Yaskawa INFORM job: A_ROOF_UPPER_0614_2_PAINT_47.JBI

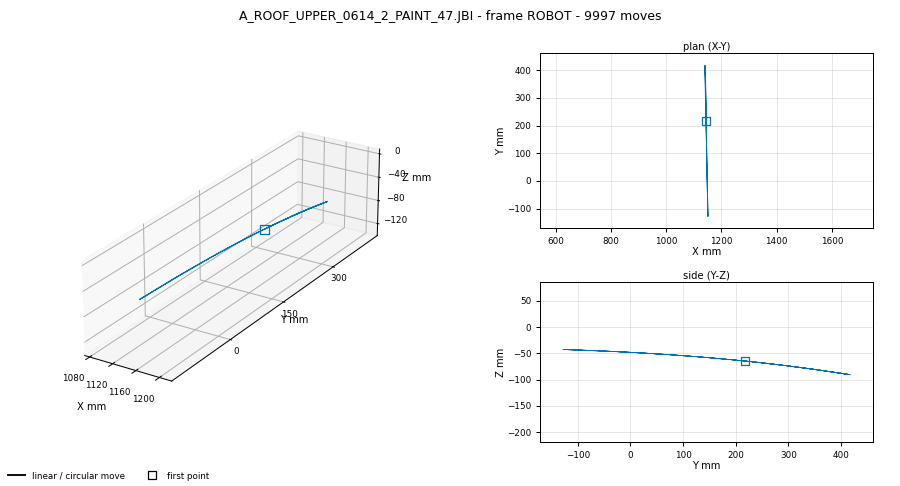
[picture p0: tool path of A_ROOF_UPPER_0614_2_PAINT_47.JBI in frame ROBOT, 9997 of 9997 moves have a stored position in this frame; points joined in program order, loops and branches not executed]
/JOB
//NAME A_ROOF_UPPER_0614_2_PAINT47
//POS
///NPOS 9997,0,0,0,0,0
///TOOL 1
///USER 0
///POSTYPE ROBOT
///RECTAN
///RCONF 1,0,0,0,0,0,0,0,0,0,0,0,0,0,0,0,0,0,0,0,0,0,0,0
C00000=1145.413,218.095,-64.507,-177.907,7.562,148.827
C00001=1145.408,218.343,-64.532,-177.904,7.565,148.827
C00002=1145.404,218.592,-64.557,-177.901,7.567,148.827
C00003=1145.399,218.840,-64.583,-177.899,7.570,148.827
C00004=1145.395,219.089,-64.609,-177.896,7.572,148.827
C00005=1145.391,219.338,-64.634,-177.893,7.575,148.827
C00006=1145.385,219.587,-64.659,-177.890,7.578,148.826
C00007=1145.381,219.835,-64.685,-177.888,7.580,148.826
C00008=1145.377,220.084,-64.711,-177.885,7.583,148.826
C00009=1145.372,220.332,-64.736,-177.882,7.586,148.826
C00010=1145.368,220.581,-64.762,-177.879,7.588,148.826
C00011=1145.364,220.830,-64.787,-177.877,7.591,148.825
C00012=1145.359,221.079,-64.812,-177.874,7.593,148.825
C00013=1145.354,221.327,-64.838,-177.871,7.596,148.825
C00014=1145.350,221.576,-64.864,-177.868,7.599,148.825
C00015=1145.345,221.824,-64.889,-177.865,7.602,148.825
C00016=1145.341,222.073,-64.915,-177.863,7.604,148.825
C00017=1145.337,222.322,-64.940,-177.860,7.607,148.825
C00018=1145.332,222.570,-64.966,-177.857,7.609,148.824
C00019=1145.328,222.819,-64.992,-177.854,7.612,148.824
C00020=1145.324,223.068,-65.017,-177.852,7.614,148.824
C00021=1145.319,223.316,-65.043,-177.849,7.617,148.824
C00022=1145.314,223.565,-65.068,-177.846,7.620,148.824
C00023=1145.310,223.813,-65.094,-177.843,7.623,148.824
C00024=1145.305,224.062,-65.121,-177.840,7.626,148.824
C00025=1145.300,224.311,-65.146,-177.838,7.628,148.823
C00026=1145.296,224.559,-65.172,-177.835,7.631,148.823
C00027=1145.292,224.808,-65.197,-177.832,7.634,148.823
C00028=1145.287,225.056,-65.223,-177.829,7.636,148.823
C00029=1145.283,225.305,-65.249,-177.826,7.639,148.823
C00030=1145.278,225.554,-65.275,-177.824,7.641,148.823
C00031=1145.274,225.803,-65.301,-177.821,7.644,148.823
C00032=1145.270,226.051,-65.327,-177.818,7.647,148.823
C00033=1145.265,226.299,-65.353,-177.815,7.650,148.822
C00034=1145.261,226.548,-65.378,-177.812,7.653,148.822
C00035=1145.256,226.797,-65.405,-177.809,7.656,148.822
C00036=1145.252,227.046,-65.430,-177.807,7.658,148.822
C00037=1145.247,227.294,-65.456,-177.804,7.661,148.822
C00038=1145.243,227.542,-65.482,-177.801,7.663,148.822
C00039=1145.239,227.791,-65.508,-177.798,7.666,148.822
C00040=1145.234,228.040,-65.534,-177.796,7.669,148.821
C00041=1145.229,228.289,-65.560,-177.793,7.671,148.821
C00042=1145.226,228.537,-65.587,-177.791,7.674,148.821
C00043=1145.220,228.786,-65.613,-177.788,7.677,148.821
C00044=1145.216,229.034,-65.638,-177.785,7.679,148.821
C00045=1145.212,229.283,-65.665,-177.782,7.682,148.821
C00046=1145.208,229.531,-65.691,-177.779,7.685,148.821
C00047=1145.203,229.781,-65.717,-177.776,7.688,148.821
C00048=1145.199,230.029,-65.743,-177.774,7.690,148.820
C00049=1145.194,230.277,-65.769,-177.771,7.693,148.820
C00050=1145.189,230.526,-65.795,-177.768,7.696,148.820
C00051=1145.185,230.774,-65.822,-177.765,7.699,148.820
C00052=1145.181,231.023,-65.847,-177.762,7.702,148.820
C00053=1145.176,231.272,-65.874,-177.760,7.705,148.820
C00054=1145.172,231.520,-65.900,-177.757,7.707,148.820
C00055=1145.167,231.769,-65.926,-177.755,7.710,148.820
C00056=1145.163,232.018,-65.953,-177.752,7.713,148.820
C00057=1145.158,232.266,-65.978,-177.748,7.715,148.819
C00058=1145.154,232.514,-66.005,-177.746,7.718,148.819
C00059=1145.149,232.763,-66.031,-177.743,7.721,148.819
C00060=1145.145,233.011,-66.058,-177.740,7.724,148.819
C00061=1145.140,233.260,-66.084,-177.738,7.726,148.819
C00062=1145.136,233.509,-66.111,-177.735,7.729,148.819
C00063=1145.132,233.758,-66.137,-177.732,7.732,148.819
C00064=1145.128,234.006,-66.163,-177.730,7.735,148.819
C00065=1145.123,234.255,-66.190,-177.726,7.737,148.818
C00066=1145.119,234.503,-66.216,-177.723,7.740,148.818
C00067=1145.114,234.751,-66.243,-177.721,7.743,148.818
C00068=1145.110,235.000,-66.269,-177.718,7.746,148.818
C00069=1145.105,235.272,-66.298,-177.715,7.749,148.818
C00070=1145.099,235.544,-66.327,-177.712,7.752,148.818
C00071=1145.095,235.815,-66.356,-177.709,7.754,148.818
C00072=1145.090,236.088,-66.385,-177.706,7.758,148.818
C00073=1145.086,236.336,-66.412,-177.703,7.760,148.817
C00074=1145.082,236.585,-66.438,-177.701,7.763,148.817
C00075=1145.077,236.834,-66.465,-177.698,7.766,148.817
C00076=1145.073,237.082,-66.492,-177.695,7.769,148.817
C00077=1145.068,237.331,-66.518,-177.692,7.772,148.817
C00078=1145.064,237.579,-66.544,-177.689,7.775,148.817
C00079=1145.059,237.827,-66.571,-177.687,7.778,148.817
C00080=1145.055,238.076,-66.599,-177.684,7.781,148.817
C00081=1145.051,238.325,-66.624,-177.681,7.783,148.817
C00082=1145.046,238.573,-66.651,-177.678,7.785,148.816
C00083=1145.041,238.822,-66.678,-177.676,7.788,148.816
C00084=1145.037,239.070,-66.705,-177.673,7.791,148.816
C00085=1145.033,239.318,-66.732,-177.670,7.794,148.816
C00086=1145.028,239.567,-66.759,-177.667,7.797,148.816
C00087=1145.024,239.816,-66.785,-177.664,7.800,148.816
C00088=1145.019,240.064,-66.812,-177.662,7.803,148.816
C00089=1145.014,240.313,-66.839,-177.659,7.806,148.816
C00090=1145.011,240.561,-66.865,-177.656,7.809,148.816
C00091=1145.006,240.809,-66.892,-177.653,7.812,148.816
C00092=1145.002,241.059,-66.920,-177.651,7.815,148.816
C00093=1144.998,241.307,-66.946,-177.648,7.818,148.816
C00094=1144.993,241.555,-66.973,-177.646,7.820,148.816
C00095=1144.989,241.804,-67.000,-177.643,7.823,148.815
C00096=1144.984,242.052,-67.028,-177.640,7.826,148.815
C00097=1144.980,242.300,-67.054,-177.637,7.828,148.815
C00098=1144.975,242.549,-67.081,-177.634,7.831,148.815
C00099=1144.971,242.797,-67.108,-177.631,7.834,148.815
C00100=1144.967,243.047,-67.136,-177.628,7.837,148.815
C00101=1144.962,243.295,-67.163,-177.626,7.840,148.815
C00102=1144.958,243.543,-67.189,-177.623,7.843,148.815
C00103=1144.953,243.792,-67.216,-177.620,7.846,148.815
C00104=1144.949,244.040,-67.243,-177.617,7.849,148.815
C00105=1144.944,244.289,-67.270,-177.614,7.852,148.814
C00106=1144.940,244.537,-67.298,-177.612,7.854,148.814
C00107=1144.936,244.786,-67.325,-177.609,7.857,148.814
C00108=1144.932,245.034,-67.352,-177.606,7.860,148.814
C00109=1144.927,245.283,-67.379,-177.603,7.863,148.814
C00110=1144.922,245.531,-67.406,-177.601,7.865,148.814
C00111=1144.918,245.780,-67.433,-177.598,7.868,148.814
C00112=1144.914,246.028,-67.461,-177.595,7.871,148.814
C00113=1144.909,246.277,-67.488,-177.593,7.874,148.814
C00114=1144.905,246.525,-67.515,-177.590,7.877,148.814
C00115=1144.900,246.774,-67.542,-177.587,7.880,148.814
C00116=1144.896,247.022,-67.569,-177.584,7.883,148.814
C00117=1144.892,247.270,-67.597,-177.581,7.886,148.814
C00118=1144.888,247.519,-67.624,-177.579,7.889,148.813
C00119=1144.883,247.767,-67.651,-177.576,7.892,148.813
C00120=1144.879,248.015,-67.679,-177.573,7.895,148.813
C00121=1144.875,248.264,-67.706,-177.570,7.897,148.813
C00122=1144.870,248.513,-67.733,-177.568,7.900,148.813
C00123=1144.866,248.761,-67.761,-177.565,7.903,148.813
C00124=1144.861,249.009,-67.788,-177.562,7.906,148.813
C00125=1144.857,249.259,-67.816,-177.559,7.909,148.813
C00126=1144.853,249.506,-67.843,-177.556,7.912,148.813
C00127=1144.848,249.755,-67.871,-177.554,7.915,148.813
C00128=1144.844,250.003,-67.899,-177.551,7.918,148.813
C00129=1144.840,250.252,-67.926,-177.548,7.921,148.813
C00130=1144.835,250.500,-67.953,-177.546,7.924,148.813
C00131=1144.831,250.748,-67.981,-177.543,7.927,148.813
C00132=1144.827,250.998,-68.008,-177.540,7.930,148.813
C00133=1144.822,251.245,-68.036,-177.537,7.933,148.813
C00134=1144.817,251.494,-68.063,-177.535,7.936,148.813
C00135=1144.813,251.743,-68.092,-177.532,7.939,148.812
C00136=1144.808,251.991,-68.119,-177.529,7.942,148.812
C00137=1144.804,252.239,-68.146,-177.526,7.945,148.812
C00138=1144.800,252.488,-68.175,-177.523,7.948,148.812
C00139=1144.796,252.736,-68.202,-177.521,7.950,148.812
C00140=1144.791,252.984,-68.229,-177.518,7.953,148.812
C00141=1144.787,253.233,-68.257,-177.515,7.956,148.812
C00142=1144.783,253.481,-68.285,-177.512,7.959,148.812
C00143=1144.778,253.730,-68.313,-177.509,7.962,148.812
C00144=1144.774,253.979,-68.340,-177.507,7.965,148.812
C00145=1144.769,254.226,-68.368,-177.504,7.968,148.812
C00146=1144.766,254.475,-68.396,-177.501,7.971,148.812
C00147=1144.761,254.724,-68.423,-177.499,7.974,148.812
C00148=1144.756,254.972,-68.452,-177.496,7.977,148.812
C00149=1144.752,255.220,-68.480,-177.493,7.980,148.812
C00150=1144.747,255.469,-68.507,-177.490,7.983,148.812
C00151=1144.744,255.717,-68.535,-177.488,7.986,148.812
C00152=1144.739,255.966,-68.563,-177.485,7.989,148.812
C00153=1144.735,256.214,-68.592,-177.482,7.992,148.811
C00154=1144.730,256.463,-68.619,-177.479,7.995,148.811
C00155=1144.726,256.710,-68.646,-177.476,7.998,148.811
C00156=1144.721,256.959,-68.675,-177.474,8.001,148.811
C00157=1144.717,257.207,-68.703,-177.471,8.004,148.811
C00158=1144.713,257.456,-68.731,-177.469,8.007,148.811
C00159=1144.709,257.704,-68.758,-177.466,8.010,148.811
C00160=1144.704,257.953,-68.787,-177.463,8.013,148.811
C00161=1144.700,258.201,-68.815,-177.460,8.015,148.811
C00162=1144.696,258.450,-68.843,-177.457,8.018,148.811
C00163=1144.691,258.698,-68.871,-177.455,8.021,148.811
C00164=1144.687,258.946,-68.899,-177.452,8.024,148.811
C00165=1144.683,259.194,-68.927,-177.449,8.028,148.811
C00166=1144.678,259.443,-68.956,-177.447,8.030,148.811
C00167=1144.674,259.691,-68.984,-177.444,8.033,148.811
C00168=1144.669,259.940,-69.012,-177.441,8.036,148.811
C00169=1144.665,260.188,-69.040,-177.438,8.039,148.811
C00170=1144.661,260.436,-69.068,-177.436,8.042,148.811
C00171=1144.656,260.685,-69.097,-177.432,8.046,148.811
C00172=1144.653,260.933,-69.125,-177.430,8.049,148.811
C00173=1144.647,261.207,-69.156,-177.427,8.052,148.811
C00174=1144.642,261.480,-69.187,-177.424,8.056,148.811
C00175=1144.638,261.753,-69.217,-177.421,8.059,148.811
C00176=1144.633,262.028,-69.249,-177.418,8.062,148.811
C00177=1144.629,262.275,-69.278,-177.415,8.065,148.811
C00178=1144.624,262.524,-69.306,-177.412,8.068,148.811
C00179=1144.620,262.772,-69.334,-177.409,8.071,148.811
C00180=1144.616,263.021,-69.363,-177.406,8.074,148.810
C00181=1144.611,263.269,-69.391,-177.404,8.077,148.811
C00182=1144.607,263.518,-69.419,-177.401,8.080,148.811
C00183=1144.603,263.766,-69.447,-177.398,8.083,148.811
C00184=1144.598,264.014,-69.477,-177.396,8.086,148.810
C00185=1144.595,264.262,-69.505,-177.393,8.089,148.810
C00186=1144.589,264.510,-69.533,-177.391,8.092,148.811
C00187=1144.586,264.759,-69.561,-177.388,8.095,148.810
C00188=1144.581,265.008,-69.590,-177.385,8.098,148.810
C00189=1144.576,265.255,-69.619,-177.382,8.101,148.810
C00190=1144.573,265.504,-69.647,-177.379,8.104,148.810
C00191=1144.568,265.752,-69.676,-177.377,8.108,148.810
C00192=1144.564,266.000,-69.704,-177.374,8.111,148.810
C00193=1144.560,266.249,-69.733,-177.371,8.114,148.810
C00194=1144.555,266.497,-69.762,-177.368,8.117,148.810
C00195=1144.551,266.745,-69.790,-177.365,8.120,148.810
C00196=1144.547,266.994,-69.819,-177.363,8.123,148.810
C00197=1144.542,267.242,-69.847,-177.360,8.126,148.810
C00198=1144.538,267.490,-69.876,-177.357,8.129,148.810
C00199=1144.534,267.739,-69.905,-177.355,8.132,148.810
C00200=1144.529,267.987,-69.933,-177.352,8.135,148.810
C00201=1144.525,268.235,-69.962,-177.350,8.138,148.810
C00202=1144.521,268.484,-69.991,-177.346,8.142,148.810
C00203=1144.516,268.732,-70.020,-177.343,8.145,148.810
C00204=1144.512,268.980,-70.048,-177.341,8.148,148.810
C00205=1144.508,269.229,-70.078,-177.338,8.151,148.810
C00206=1144.503,269.477,-70.106,-177.336,8.154,148.810
C00207=1144.499,269.725,-70.135,-177.333,8.157,148.810
C00208=1144.495,269.974,-70.164,-177.330,8.160,148.810
C00209=1144.491,270.222,-70.193,-177.328,8.163,148.810
C00210=1144.486,270.471,-70.222,-177.325,8.166,148.810
C00211=1144.482,270.718,-70.250,-177.321,8.170,148.810
C00212=1144.478,270.967,-70.279,-177.319,8.173,148.810
C00213=1144.473,271.215,-70.309,-177.316,8.176,148.810
C00214=1144.469,271.463,-70.338,-177.314,8.179,148.810
C00215=1144.464,271.712,-70.366,-177.311,8.182,148.810
C00216=1144.461,271.960,-70.395,-177.308,8.185,148.810
C00217=1144.457,272.208,-70.425,-177.306,8.188,148.810
C00218=1144.452,272.457,-70.453,-177.303,8.191,148.810
C00219=1144.447,272.704,-70.483,-177.300,8.194,148.810
C00220=1144.443,272.953,-70.512,-177.297,8.198,148.810
C00221=1144.439,273.201,-70.541,-177.294,8.201,148.810
C00222=1144.434,273.450,-70.570,-177.292,8.204,148.810
C00223=1144.431,273.698,-70.599,-177.289,8.207,148.810
C00224=1144.426,273.946,-70.627,-177.287,8.210,148.810
C00225=1144.422,274.194,-70.657,-177.284,8.213,148.810
C00226=1144.418,274.442,-70.686,-177.281,8.216,148.811
C00227=1144.413,274.691,-70.716,-177.278,8.220,148.811
C00228=1144.409,274.939,-70.745,-177.275,8.223,148.810
C00229=1144.405,275.188,-70.774,-177.273,8.226,148.811
C00230=1144.401,275.436,-70.803,-177.270,8.229,148.811
C00231=1144.396,275.684,-70.833,-177.267,8.232,148.811
C00232=1144.392,275.932,-70.862,-177.265,8.235,148.810
C00233=1144.387,276.180,-70.891,-177.262,8.238,148.811
C00234=1144.383,276.428,-70.921,-177.259,8.242,148.811
C00235=1144.379,276.677,-70.950,-177.256,8.245,148.811
C00236=1144.376,276.925,-70.979,-177.254,8.248,148.811
C00237=1144.371,277.174,-71.008,-177.251,8.251,148.811
C00238=1144.367,277.422,-71.037,-177.248,8.254,148.811
C00239=1144.362,277.669,-71.066,-177.246,8.257,148.811
C00240=1144.357,277.918,-71.097,-177.243,8.261,148.811
C00241=1144.353,278.166,-71.126,-177.240,8.264,148.811
C00242=1144.349,278.414,-71.155,-177.237,8.267,148.811
C00243=1144.345,278.663,-71.185,-177.235,8.270,148.811
C00244=1144.340,278.911,-71.214,-177.232,8.273,148.811
C00245=1144.336,279.159,-71.244,-177.229,8.276,148.811
C00246=1144.332,279.408,-71.273,-177.226,8.280,148.811
C00247=1144.328,279.656,-71.303,-177.224,8.283,148.811
C00248=1144.324,279.903,-71.333,-177.221,8.286,148.811
C00249=1144.320,280.152,-71.362,-177.218,8.289,148.811
C00250=1144.316,280.400,-71.392,-177.216,8.293,148.811
C00251=1144.312,280.648,-71.421,-177.213,8.295,148.811
C00252=1144.307,280.897,-71.451,-177.210,8.300,148.811
C00253=1144.302,281.145,-71.481,-177.207,8.302,148.811
C00254=1144.298,281.393,-71.510,-177.205,8.305,148.811
C00255=1144.294,281.642,-71.540,-177.202,8.309,148.811
C00256=1144.290,281.889,-71.570,-177.200,8.312,148.811
C00257=1144.286,282.138,-71.599,-177.197,8.316,148.812
C00258=1144.281,282.386,-71.629,-177.194,8.319,148.811
C00259=1144.277,282.634,-71.659,-177.191,8.322,148.811
C00260=1144.273,282.882,-71.689,-177.189,8.325,148.812
C00261=1144.269,283.130,-71.718,-177.186,8.328,148.812
C00262=1144.265,283.379,-71.748,-177.184,8.331,148.812
C00263=1144.260,283.627,-71.778,-177.180,8.335,148.812
C00264=1144.256,283.875,-71.808,-177.178,8.338,148.812
C00265=1144.252,284.123,-71.837,-177.175,8.341,148.812
C00266=1144.248,284.371,-71.867,-177.172,8.344,148.812
C00267=1144.243,284.619,-71.898,-177.170,8.347,148.812
C00268=1144.239,284.868,-71.927,-177.167,8.351,148.812
C00269=1144.235,285.116,-71.957,-177.164,8.354,148.812
C00270=1144.230,285.364,-71.987,-177.162,8.357,148.812
C00271=1144.226,285.612,-72.017,-177.159,8.360,148.812
C00272=1144.222,285.860,-72.047,-177.156,8.364,148.812
C00273=1144.217,286.108,-72.077,-177.154,8.367,148.812
C00274=1144.213,286.357,-72.106,-177.151,8.370,148.812
C00275=1144.209,286.604,-72.137,-177.148,8.373,148.812
C00276=1144.205,286.854,-72.167,-177.146,8.376,148.812
C00277=1144.200,287.128,-72.200,-177.142,8.380,148.812
C00278=1144.195,287.403,-72.234,-177.139,8.384,148.813
C00279=1144.191,287.679,-72.267,-177.137,8.387,148.813
C00280=1144.186,287.954,-72.301,-177.134,8.391,148.813
C00281=1144.182,288.203,-72.330,-177.131,8.394,148.813
C00282=1144.177,288.451,-72.361,-177.128,8.398,148.813
C00283=1144.173,288.699,-72.391,-177.125,8.401,148.813
C00284=1144.169,288.947,-72.421,-177.123,8.405,148.813
C00285=1144.165,289.195,-72.452,-177.120,8.407,148.813
C00286=1144.161,289.443,-72.481,-177.117,8.412,148.813
C00287=1144.156,289.691,-72.512,-177.114,8.415,148.813
C00288=1144.153,289.940,-72.542,-177.112,8.418,148.813
C00289=1144.148,290.188,-72.572,-177.109,8.421,148.813
C00290=1144.144,290.436,-72.603,-177.107,8.424,148.814
C00291=1144.139,290.684,-72.633,-177.104,8.428,148.814
C00292=1144.135,290.932,-72.663,-177.101,8.431,148.814
C00293=1144.131,291.181,-72.694,-177.098,8.434,148.814
C00294=1144.127,291.428,-72.724,-177.096,8.437,148.814
C00295=1144.123,291.676,-72.755,-177.093,8.441,148.814
C00296=1144.118,291.925,-72.784,-177.090,8.444,148.814
C00297=1144.114,292.173,-72.815,-177.088,8.447,148.814
C00298=1144.110,292.421,-72.846,-177.085,8.450,148.814
C00299=1144.106,292.669,-72.876,-177.082,8.454,148.814
C00300=1144.102,292.916,-72.907,-177.080,8.457,148.814
C00301=1144.097,293.165,-72.937,-177.077,8.461,148.814
C00302=1144.094,293.413,-72.967,-177.075,8.464,148.814
C00303=1144.089,293.661,-72.998,-177.072,8.468,148.815
C00304=1144.085,293.909,-73.029,-177.069,8.471,148.815
C00305=1144.081,294.157,-73.059,-177.066,8.474,148.815
C00306=1144.077,294.406,-73.090,-177.063,8.478,148.815
C00307=1144.072,294.654,-73.121,-177.061,8.481,148.815
C00308=1144.068,294.901,-73.151,-177.058,8.484,148.815
C00309=1144.064,295.150,-73.182,-177.056,8.487,148.815
C00310=1144.060,295.398,-73.212,-177.053,8.491,148.815
C00311=1144.056,295.645,-73.243,-177.050,8.494,148.815
C00312=1144.051,295.894,-73.273,-177.048,8.497,148.815
C00313=1144.047,296.142,-73.303,-177.045,8.501,148.816
C00314=1144.043,296.390,-73.335,-177.042,8.504,148.816
C00315=1144.039,296.638,-73.366,-177.040,8.508,148.816
C00316=1144.035,296.886,-73.397,-177.037,8.511,148.816
C00317=1144.031,297.134,-73.427,-177.034,8.515,148.816
C00318=1144.026,297.382,-73.458,-177.032,8.518,148.816
C00319=1144.022,297.631,-73.489,-177.029,8.521,148.816
C00320=1144.018,297.878,-73.519,-177.026,8.524,148.816
C00321=1144.014,298.126,-73.550,-177.023,8.528,148.816
C00322=1144.010,298.375,-73.581,-177.021,8.531,148.816
C00323=1144.005,298.623,-73.612,-177.018,8.534,148.817
C00324=1144.001,298.872,-73.643,-177.015,8.538,148.817
C00325=1143.997,299.119,-73.674,-177.013,8.541,148.817
C00326=1143.993,299.366,-73.705,-177.010,8.545,148.817
C00327=1143.989,299.615,-73.736,-177.007,8.548,148.817
C00328=1143.984,299.863,-73.766,-177.005,8.552,148.817
C00329=1143.980,300.111,-73.797,-177.002,8.555,148.817
C00330=1143.976,300.359,-73.829,-177.000,8.558,148.817
C00331=1143.972,300.607,-73.859,-176.997,8.562,148.818
C00332=1143.968,300.855,-73.890,-176.994,8.565,148.818
C00333=1143.964,301.103,-73.922,-176.992,8.568,148.818
C00334=1143.960,301.351,-73.953,-176.989,8.572,148.818
C00335=1143.955,301.599,-73.984,-176.986,8.576,148.818
C00336=1143.950,301.847,-74.014,-176.984,8.578,148.818
C00337=1143.947,302.095,-74.046,-176.981,8.583,148.818
C00338=1143.942,302.343,-74.077,-176.978,8.586,148.818
C00339=1143.938,302.591,-74.109,-176.976,8.589,148.818
C00340=1143.934,302.839,-74.140,-176.973,8.593,148.819
C00341=1143.930,303.088,-74.170,-176.970,8.596,148.819
C00342=1143.926,303.335,-74.202,-176.968,8.599,148.819
C00343=1143.922,303.583,-74.232,-176.965,8.603,148.819
C00344=1143.918,303.831,-74.264,-176.962,8.606,148.819
C00345=1143.913,304.079,-74.295,-176.960,8.610,148.819
C00346=1143.909,304.328,-74.326,-176.957,8.613,148.819
C00347=1143.905,304.575,-74.358,-176.954,8.617,148.819
C00348=1143.901,304.824,-74.389,-176.952,8.620,148.820
C00349=1143.897,305.071,-74.420,-176.949,8.624,148.820
C00350=1143.893,305.320,-74.451,-176.946,8.627,148.820
C00351=1143.888,305.567,-74.483,-176.944,8.630,148.820
C00352=1143.884,305.815,-74.515,-176.941,8.634,148.820
C00353=1143.879,306.063,-74.546,-176.939,8.638,148.820
C00354=1143.875,306.311,-74.578,-176.936,8.640,148.820
C00355=1143.871,306.559,-74.609,-176.933,8.645,148.821
C00356=1143.867,306.807,-74.641,-176.931,8.648,148.821
C00357=1143.863,307.055,-74.672,-176.928,8.651,148.821
C00358=1143.859,307.303,-74.703,-176.925,8.655,148.821
C00359=1143.855,307.551,-74.735,-176.923,8.658,148.821
C00360=1143.851,307.799,-74.766,-176.920,8.661,148.821
C00361=1143.847,308.047,-74.798,-176.917,8.665,148.822
C00362=1143.843,308.295,-74.829,-176.915,8.669,148.822
C00363=1143.838,308.543,-74.862,-176.912,8.672,148.822
C00364=1143.834,308.792,-74.893,-176.909,8.676,148.822
C00365=1143.830,309.039,-74.924,-176.907,8.679,148.822
C00366=1143.826,309.287,-74.956,-176.904,8.683,148.822
C00367=1143.822,309.534,-74.987,-176.901,8.686,148.822
C00368=1143.818,309.783,-75.019,-176.899,8.689,148.822
C00369=1143.813,310.031,-75.051,-176.896,8.693,148.823
C00370=1143.809,310.279,-75.083,-176.894,8.697,148.823
C00371=1143.805,310.527,-75.114,-176.891,8.700,148.823
C00372=1143.801,310.774,-75.146,-176.888,8.704,148.823
C00373=1143.797,311.022,-75.178,-176.886,8.707,148.823
C00374=1143.793,311.271,-75.209,-176.883,8.711,148.823
C00375=1143.788,311.518,-75.241,-176.880,8.714,148.824
C00376=1143.784,311.767,-75.273,-176.878,8.718,148.824
C00377=1143.780,312.015,-75.305,-176.875,8.722,148.824
C00378=1143.776,312.262,-75.337,-176.873,8.725,148.824
C00379=1143.772,312.510,-75.369,-176.869,8.729,148.824
C00380=1143.768,312.758,-75.400,-176.867,8.732,148.824
C00381=1143.763,313.036,-75.437,-176.864,8.736,148.825
C00382=1143.759,313.314,-75.472,-176.861,8.740,148.825
C00383=1143.754,313.591,-75.508,-176.858,8.744,148.825
C00384=1143.749,313.870,-75.543,-176.855,8.748,148.825
C00385=1143.746,314.117,-75.576,-176.853,8.751,148.826
C00386=1143.741,314.365,-75.608,-176.850,8.754,148.826
C00387=1143.737,314.613,-75.640,-176.847,8.758,148.826
C00388=1143.733,314.861,-75.672,-176.845,8.762,148.826
C00389=1143.729,315.109,-75.704,-176.842,8.766,148.826
C00390=1143.725,315.356,-75.736,-176.840,8.769,148.826
C00391=1143.720,315.605,-75.768,-176.838,8.772,148.827
C00392=1143.717,315.853,-75.800,-176.835,8.776,148.827
C00393=1143.712,316.100,-75.831,-176.832,8.780,148.827
C00394=1143.708,316.348,-75.864,-176.829,8.784,148.827
C00395=1143.704,316.596,-75.896,-176.827,8.787,148.827
C00396=1143.700,316.844,-75.929,-176.824,8.790,148.827
C00397=1143.696,317.092,-75.961,-176.821,8.794,148.828
C00398=1143.691,317.340,-75.993,-176.819,8.797,148.828
C00399=1143.688,317.587,-76.025,-176.816,8.801,148.828
C00400=1143.684,317.835,-76.057,-176.814,8.805,148.828
C00401=1143.680,318.084,-76.089,-176.811,8.809,148.828
C00402=1143.676,318.332,-76.121,-176.809,8.812,148.829
C00403=1143.671,318.579,-76.154,-176.806,8.815,148.829
C00404=1143.667,318.827,-76.186,-176.803,8.819,148.829
C00405=1143.663,319.075,-76.218,-176.801,8.823,148.829
C00406=1143.660,319.323,-76.251,-176.798,8.827,148.829
C00407=1143.655,319.571,-76.283,-176.796,8.830,148.830
C00408=1143.651,319.819,-76.316,-176.793,8.834,148.830
C00409=1143.647,320.066,-76.348,-176.790,8.837,148.830
C00410=1143.642,320.314,-76.380,-176.787,8.841,148.830
C00411=1143.639,320.562,-76.413,-176.785,8.845,148.830
C00412=1143.634,320.810,-76.445,-176.783,8.848,148.831
C00413=1143.631,321.058,-76.478,-176.780,8.852,148.831
C00414=1143.627,321.306,-76.510,-176.778,8.855,148.831
C00415=1143.622,321.554,-76.544,-176.775,8.859,148.831
C00416=1143.618,321.801,-76.575,-176.772,8.863,148.831
C00417=1143.614,322.049,-76.608,-176.769,8.867,148.832
C00418=1143.610,322.297,-76.640,-176.767,8.870,148.832
C00419=1143.606,322.545,-76.673,-176.764,8.874,148.832
C00420=1143.602,322.793,-76.706,-176.762,8.877,148.832
C00421=1143.598,323.040,-76.738,-176.759,8.881,148.832
C00422=1143.594,323.289,-76.771,-176.757,8.885,148.833
C00423=1143.590,323.536,-76.804,-176.754,8.888,148.833
C00424=1143.586,323.784,-76.836,-176.751,8.892,148.833
C00425=1143.582,324.032,-76.869,-176.749,8.895,148.833
C00426=1143.578,324.280,-76.902,-176.746,8.899,148.834
C00427=1143.574,324.528,-76.934,-176.744,8.903,148.834
C00428=1143.570,324.776,-76.967,-176.741,8.907,148.834
C00429=1143.566,325.023,-77.000,-176.738,8.910,148.834
C00430=1143.561,325.271,-77.032,-176.736,8.914,148.834
C00431=1143.557,325.518,-77.065,-176.733,8.917,148.835
C00432=1143.553,325.766,-77.098,-176.730,8.921,148.835
C00433=1143.549,326.014,-77.131,-176.728,8.925,148.835
C00434=1143.545,326.262,-77.164,-176.725,8.929,148.835
C00435=1143.540,326.510,-77.197,-176.723,8.932,148.835
C00436=1143.537,326.757,-77.229,-176.720,8.936,148.836
C00437=1143.533,327.005,-77.262,-176.718,8.940,148.836
C00438=1143.528,327.253,-77.295,-176.715,8.944,148.836
C00439=1143.524,327.501,-77.328,-176.713,8.947,148.836
C00440=1143.520,327.749,-77.361,-176.710,8.951,148.837
C00441=1143.516,327.997,-77.394,-176.707,8.954,148.837
C00442=1143.513,328.244,-77.427,-176.704,8.958,148.837
C00443=1143.509,328.492,-77.460,-176.702,8.962,148.837
C00444=1143.504,328.740,-77.493,-176.699,8.966,148.838
C00445=1143.500,328.987,-77.526,-176.697,8.969,148.838
C00446=1143.496,329.236,-77.559,-176.694,8.973,148.838
C00447=1143.492,329.484,-77.592,-176.692,8.977,148.838
C00448=1143.488,329.732,-77.625,-176.689,8.981,148.839
C00449=1143.484,329.980,-77.659,-176.687,8.984,148.839
C00450=1143.480,330.227,-77.692,-176.684,8.988,148.839
C00451=1143.476,330.475,-77.725,-176.682,8.991,148.839
C00452=1143.472,330.723,-77.758,-176.679,8.995,148.839
C00453=1143.468,330.970,-77.791,-176.677,8.999,148.840
C00454=1143.464,331.218,-77.824,-176.674,9.003,148.840
C00455=1143.460,331.466,-77.857,-176.671,9.006,148.840
C00456=1143.456,331.713,-77.891,-176.669,9.010,148.841
C00457=1143.452,331.960,-77.924,-176.666,9.014,148.841
C00458=1143.448,332.208,-77.957,-176.663,9.018,148.841
C00459=1143.444,332.457,-77.991,-176.661,9.021,148.841
C00460=1143.440,332.704,-78.024,-176.658,9.025,148.842
C00461=1143.436,332.952,-78.057,-176.656,9.029,148.842
C00462=1143.431,333.200,-78.091,-176.653,9.033,148.842
C00463=1143.427,333.448,-78.124,-176.651,9.036,148.842
C00464=1143.423,333.695,-78.158,-176.648,9.040,148.842
C00465=1143.419,333.943,-78.191,-176.646,9.044,148.843
C00466=1143.415,334.191,-78.224,-176.643,9.048,148.843
C00467=1143.411,334.439,-78.258,-176.641,9.051,148.843
C00468=1143.408,334.686,-78.291,-176.638,9.055,148.844
C00469=1143.403,334.934,-78.325,-176.635,9.059,148.844
C00470=1143.399,335.181,-78.358,-176.633,9.063,148.844
C00471=1143.395,335.429,-78.391,-176.630,9.067,148.844
C00472=1143.392,335.677,-78.425,-176.628,9.070,148.845
C00473=1143.387,335.925,-78.459,-176.625,9.074,148.845
C00474=1143.383,336.173,-78.492,-176.623,9.078,148.845
C00475=1143.379,336.420,-78.526,-176.620,9.082,148.846
C00476=1143.375,336.668,-78.559,-176.618,9.085,148.846
C00477=1143.372,336.915,-78.593,-176.615,9.089,148.846
C00478=1143.368,337.163,-78.627,-176.613,9.093,148.846
C00479=1143.363,337.411,-78.660,-176.610,9.097,148.847
C00480=1143.359,337.658,-78.694,-176.607,9.101,148.847
C00481=1143.355,337.907,-78.728,-176.605,9.104,148.847
C00482=1143.351,338.154,-78.762,-176.602,9.109,148.848
C00483=1143.347,338.401,-78.795,-176.600,9.112,148.848
C00484=1143.343,338.649,-78.829,-176.597,9.116,148.848
C00485=1143.339,338.929,-78.867,-176.594,9.120,148.848
C00486=1143.334,339.210,-78.906,-176.592,9.124,148.849
C00487=1143.329,339.491,-78.943,-176.589,9.128,148.849
C00488=1143.325,339.771,-78.981,-176.585,9.133,148.849
C00489=1143.320,340.019,-79.016,-176.583,9.137,148.850
C00490=1143.317,340.267,-79.050,-176.580,9.141,148.850
C00491=1143.313,340.514,-79.083,-176.578,9.144,148.850
C00492=1143.308,340.762,-79.118,-176.575,9.149,148.850
C00493=1143.305,341.010,-79.151,-176.573,9.152,148.851
C00494=1143.301,341.257,-79.185,-176.570,9.156,148.851
C00495=1143.296,341.505,-79.219,-176.568,9.160,148.851
C00496=1143.293,341.753,-79.253,-176.565,9.164,148.852
C00497=1143.288,342.001,-79.287,-176.562,9.168,148.852
C00498=1143.285,342.248,-79.321,-176.561,9.171,148.852
C00499=1143.280,342.495,-79.354,-176.558,9.175,148.852
C00500=1143.276,342.743,-79.389,-176.555,9.179,148.853
C00501=1143.273,342.991,-79.423,-176.553,9.183,148.853
C00502=1143.269,343.239,-79.458,-176.550,9.187,148.853
C00503=1143.265,343.486,-79.491,-176.548,9.190,148.854
C00504=1143.261,343.734,-79.525,-176.545,9.195,148.854
C00505=1143.257,343.982,-79.560,-176.542,9.199,148.854
C00506=1143.253,344.229,-79.594,-176.540,9.202,148.854
C00507=1143.248,344.476,-79.628,-176.537,9.206,148.855
C00508=1143.245,344.724,-79.662,-176.535,9.210,148.855
C00509=1143.240,344.972,-79.696,-176.532,9.214,148.856
C00510=1143.237,345.220,-79.730,-176.530,9.218,148.856
C00511=1143.232,345.467,-79.765,-176.527,9.221,148.856
C00512=1143.229,345.714,-79.799,-176.525,9.226,148.856
C00513=1143.225,345.963,-79.834,-176.522,9.230,148.857
C00514=1143.221,346.210,-79.867,-176.520,9.234,148.857
C00515=1143.217,346.458,-79.902,-176.517,9.238,148.857
C00516=1143.213,346.705,-79.936,-176.515,9.241,148.858
C00517=1143.208,346.952,-79.971,-176.512,9.245,148.858
C00518=1143.204,347.200,-80.005,-176.509,9.249,148.858
C00519=1143.201,347.447,-80.039,-176.507,9.253,148.859
C00520=1143.197,347.696,-80.074,-176.504,9.257,148.859
C00521=1143.193,347.943,-80.108,-176.501,9.261,148.859
C00522=1143.189,348.191,-80.143,-176.500,9.265,148.860
C00523=1143.184,348.438,-80.177,-176.497,9.269,148.860
C00524=1143.181,348.686,-80.212,-176.495,9.272,148.860
C00525=1143.176,348.934,-80.246,-176.492,9.276,148.860
C00526=1143.173,349.181,-80.280,-176.489,9.281,148.861
C00527=1143.169,349.429,-80.315,-176.487,9.284,148.861
C00528=1143.165,349.676,-80.350,-176.484,9.288,148.861
C00529=1143.161,349.923,-80.384,-176.482,9.292,148.862
C00530=1143.157,350.171,-80.419,-176.479,9.296,148.862
C00531=1143.153,350.419,-80.453,-176.477,9.300,148.863
C00532=1143.149,350.667,-80.488,-176.474,9.304,148.863
C00533=1143.145,350.913,-80.523,-176.472,9.308,148.863
C00534=1143.141,351.162,-80.558,-176.469,9.312,148.863
C00535=1143.137,351.409,-80.592,-176.466,9.316,148.864
C00536=1143.133,351.657,-80.626,-176.464,9.320,148.864
C00537=1143.129,351.904,-80.662,-176.462,9.324,148.865
C00538=1143.125,352.152,-80.696,-176.459,9.328,148.865
C00539=1143.121,352.400,-80.731,-176.457,9.332,148.865
C00540=1143.118,352.646,-80.766,-176.454,9.336,148.865
C00541=1143.114,352.894,-80.801,-176.451,9.340,148.866
C00542=1143.109,353.142,-80.835,-176.449,9.343,148.866
C00543=1143.105,353.389,-80.871,-176.446,9.348,148.867
C00544=1143.102,353.637,-80.905,-176.444,9.352,148.867
C00545=1143.098,353.885,-80.939,-176.442,9.355,148.867
C00546=1143.094,354.132,-80.975,-176.439,9.359,148.867
C00547=1143.089,354.380,-81.009,-176.436,9.364,148.868
C00548=1143.086,354.627,-81.045,-176.434,9.367,148.868
C00549=1143.083,354.875,-81.079,-176.431,9.371,148.869
C00550=1143.078,355.122,-81.114,-176.428,9.376,148.869
C00551=1143.074,355.370,-81.149,-176.427,9.379,148.869
C00552=1143.070,355.617,-81.184,-176.424,9.383,148.870
C00553=1143.066,355.865,-81.219,-176.421,9.388,148.870
C00554=1143.062,356.112,-81.255,-176.419,9.391,148.870
C00555=1143.058,356.360,-81.289,-176.416,9.395,148.871
C00556=1143.054,356.607,-81.325,-176.413,9.399,148.871
C00557=1143.051,356.855,-81.359,-176.411,9.403,148.871
C00558=1143.047,357.102,-81.394,-176.409,9.407,148.872
C00559=1143.043,357.349,-81.430,-176.406,9.411,148.872
C00560=1143.039,357.597,-81.465,-176.404,9.416,148.872
C00561=1143.035,357.844,-81.500,-176.401,9.419,148.873
C00562=1143.031,358.092,-81.535,-176.399,9.423,148.873
C00563=1143.027,358.340,-81.570,-176.396,9.427,148.873
C00564=1143.023,358.587,-81.606,-176.394,9.431,148.874
C00565=1143.019,358.834,-81.641,-176.391,9.435,148.874
C00566=1143.015,359.082,-81.676,-176.388,9.440,148.875
C00567=1143.012,359.330,-81.711,-176.386,9.444,148.875
C00568=1143.008,359.577,-81.747,-176.384,9.447,148.875
C00569=1143.004,359.824,-81.782,-176.381,9.452,148.876
C00570=1143.000,360.072,-81.817,-176.378,9.456,148.876
C00571=1142.996,360.320,-81.852,-176.376,9.460,148.876
C00572=1142.992,360.567,-81.888,-176.373,9.463,148.877
C00573=1142.988,360.814,-81.923,-176.371,9.468,148.877
C00574=1142.984,361.061,-81.959,-176.368,9.472,148.877
C00575=1142.981,361.309,-81.994,-176.365,9.476,148.878
C00576=1142.977,361.557,-82.029,-176.363,9.481,148.878
C00577=1142.973,361.804,-82.064,-176.361,9.484,148.878
C00578=1142.968,362.052,-82.100,-176.358,9.488,148.879
C00579=1142.964,362.299,-82.136,-176.355,9.492,148.879
C00580=1142.961,362.547,-82.171,-176.353,9.497,148.880
C00581=1142.957,362.794,-82.207,-176.350,9.501,148.880
C00582=1142.953,363.041,-82.242,-176.347,9.505,148.880
C00583=1142.949,363.288,-82.278,-176.344,9.509,148.881
C00584=1142.946,363.536,-82.313,-176.342,9.513,148.881
C00585=1142.942,363.783,-82.349,-176.340,9.517,148.881
C00586=1142.937,364.031,-82.385,-176.337,9.521,148.882
C00587=1142.934,364.279,-82.420,-176.334,9.526,148.882
C00588=1142.930,364.526,-82.456,-176.331,9.530,148.882
C00589=1142.926,364.810,-82.497,-176.328,9.535,148.883
C00590=1142.921,365.093,-82.538,-176.326,9.539,148.883
C00591=1142.916,365.377,-82.579,-176.322,9.544,148.884
C00592=1142.912,365.660,-82.620,-176.320,9.549,148.884
C00593=1142.908,365.908,-82.655,-176.317,9.553,148.885
C00594=1142.904,366.155,-82.691,-176.314,9.557,148.885
C00595=1142.900,366.403,-82.727,-176.312,9.561,148.885
C00596=1142.897,366.650,-82.763,-176.309,9.565,148.886
C00597=1142.893,366.897,-82.799,-176.306,9.570,148.886
C00598=1142.889,367.145,-82.834,-176.304,9.574,148.886
C00599=1142.885,367.393,-82.870,-176.301,9.578,148.887
C00600=1142.882,367.639,-82.907,-176.299,9.583,148.887
C00601=1142.878,367.887,-82.942,-176.296,9.587,148.888
C00602=1142.873,368.134,-82.978,-176.293,9.591,148.888
C00603=1142.869,368.382,-83.014,-176.290,9.595,148.888
C00604=1142.866,368.628,-83.050,-176.288,9.600,148.889
C00605=1142.861,368.876,-83.086,-176.285,9.604,148.889
C00606=1142.858,369.124,-83.122,-176.282,9.608,148.890
C00607=1142.854,369.371,-83.158,-176.280,9.612,148.890
C00608=1142.850,369.618,-83.194,-176.278,9.616,148.890
C00609=1142.847,369.865,-83.230,-176.275,9.620,148.891
C00610=1142.842,370.113,-83.266,-176.272,9.624,148.891
C00611=1142.839,370.361,-83.302,-176.270,9.629,148.892
C00612=1142.835,370.608,-83.339,-176.267,9.633,148.892
C00613=1142.831,370.855,-83.374,-176.264,9.637,148.892
C00614=1142.827,371.103,-83.411,-176.262,9.642,148.893
C00615=1142.823,371.350,-83.447,-176.259,9.646,148.893
C00616=1142.819,371.597,-83.484,-176.256,9.650,148.894
C00617=1142.815,371.845,-83.519,-176.254,9.655,148.894
C00618=1142.812,372.092,-83.555,-176.251,9.659,148.895
C00619=1142.808,372.339,-83.592,-176.250,9.663,148.895
C00620=1142.804,372.586,-83.628,-176.247,9.667,148.895
C00621=1142.800,372.833,-83.665,-176.244,9.671,148.896
C00622=1142.796,373.081,-83.701,-176.242,9.675,148.896
C00623=1142.792,373.328,-83.737,-176.239,9.680,148.897
C00624=1142.788,373.575,-83.774,-176.237,9.684,148.897
C00625=1142.785,373.823,-83.809,-176.235,9.688,148.897
C00626=1142.781,374.071,-83.847,-176.232,9.692,148.898
C00627=1142.778,374.318,-83.883,-176.230,9.696,148.898
C00628=1142.773,374.565,-83.919,-176.227,9.701,148.899
C00629=1142.770,374.812,-83.955,-176.225,9.704,148.899
C00630=1142.766,375.060,-83.992,-176.223,9.709,148.900
C00631=1142.762,375.307,-84.028,-176.220,9.713,148.900
C00632=1142.758,375.554,-84.065,-176.218,9.718,148.901
C00633=1142.754,375.801,-84.102,-176.216,9.721,148.901
C00634=1142.750,376.049,-84.138,-176.213,9.726,148.902
C00635=1142.747,376.295,-84.175,-176.211,9.729,148.902
C00636=1142.743,376.544,-84.211,-176.209,9.733,148.902
C00637=1142.739,376.791,-84.248,-176.207,9.738,148.903
C00638=1142.735,377.038,-84.284,-176.205,9.742,148.904
C00639=1142.731,377.285,-84.321,-176.202,9.746,148.904
C00640=1142.727,377.532,-84.358,-176.200,9.750,148.904
C00641=1142.724,377.779,-84.394,-176.199,9.754,148.905
C00642=1142.720,378.027,-84.431,-176.196,9.758,148.906
C00643=1142.716,378.275,-84.468,-176.195,9.762,148.906
C00644=1142.713,378.522,-84.504,-176.192,9.766,148.907
C00645=1142.709,378.769,-84.541,-176.190,9.770,148.907
C00646=1142.704,379.016,-84.578,-176.189,9.774,148.908
C00647=1142.700,379.263,-84.614,-176.187,9.778,148.908
C00648=1142.697,379.510,-84.651,-176.185,9.781,148.909
C00649=1142.693,379.758,-84.688,-176.183,9.786,148.909
C00650=1142.689,380.005,-84.725,-176.181,9.789,148.910
C00651=1142.685,380.253,-84.762,-176.180,9.793,148.910
C00652=1142.681,380.500,-84.799,-176.178,9.797,148.911
C00653=1142.678,380.747,-84.835,-176.177,9.801,148.912
C00654=1142.674,380.995,-84.872,-176.176,9.804,148.912
C00655=1142.670,381.242,-84.909,-176.174,9.808,148.913
C00656=1142.666,381.489,-84.946,-176.173,9.812,148.913
C00657=1142.662,381.736,-84.983,-176.171,9.815,148.914
C00658=1142.659,381.982,-85.020,-176.170,9.818,148.914
C00659=1142.656,382.230,-85.057,-176.169,9.822,148.915
C00660=1142.651,382.478,-85.094,-176.167,9.826,148.916
C00661=1142.647,382.725,-85.130,-176.167,9.830,148.916
C00662=1142.643,382.972,-85.167,-176.166,9.833,148.917
C00663=1142.640,383.220,-85.205,-176.164,9.837,148.918
C00664=1142.636,383.467,-85.241,-176.163,9.840,148.918
C00665=1142.633,383.713,-85.278,-176.163,9.843,148.919
C00666=1142.628,383.960,-85.315,-176.162,9.846,148.919
C00667=1142.625,384.208,-85.352,-176.161,9.850,148.920
C00668=1142.621,384.456,-85.389,-176.160,9.853,148.921
C00669=1142.617,384.703,-85.426,-176.159,9.857,148.921
C00670=1142.613,384.950,-85.463,-176.160,9.859,148.922
C00671=1142.610,385.197,-85.501,-176.159,9.862,148.923
C00672=1142.606,385.444,-85.537,-176.158,9.866,148.923
C00673=1142.602,385.691,-85.574,-176.158,9.869,148.924
C00674=1142.598,385.938,-85.611,-176.158,9.872,148.925
C00675=1142.595,386.186,-85.649,-176.157,9.875,148.926
C00676=1142.591,386.433,-85.686,-176.157,9.878,148.926
C00677=1142.587,386.680,-85.723,-176.157,9.881,148.927
C00678=1142.583,386.928,-85.760,-176.157,9.884,148.928
C00679=1142.579,387.175,-85.797,-176.157,9.886,148.929
C00680=1142.575,387.422,-85.834,-176.156,9.889,148.929
C00681=1142.571,387.669,-85.871,-176.157,9.892,148.930
C00682=1142.568,387.917,-85.908,-176.157,9.895,148.931
C00683=1142.565,388.163,-85.945,-176.157,9.897,148.932
C00684=1142.561,388.410,-85.982,-176.157,9.900,148.932
C00685=1142.557,388.658,-86.019,-176.157,9.903,148.933
C00686=1142.553,388.905,-86.057,-176.158,9.905,148.934
C00687=1142.549,389.152,-86.094,-176.158,9.908,148.935
C00688=1142.546,389.400,-86.131,-176.158,9.911,148.935
C00689=1142.542,389.647,-86.168,-176.159,9.913,148.936
C00690=1142.538,389.894,-86.206,-176.160,9.916,148.937
C00691=1142.534,390.141,-86.242,-176.160,9.918,148.938
C00692=1142.530,390.389,-86.280,-176.160,9.921,148.939
C00693=1142.526,390.675,-86.323,-176.161,9.924,148.939
C00694=1142.522,390.963,-86.366,-176.162,9.926,148.940
C00695=1142.517,391.249,-86.410,-176.162,9.929,148.941
C00696=1142.513,391.537,-86.452,-176.163,9.932,148.942
C00697=1142.509,391.784,-86.489,-176.164,9.934,148.943
C00698=1142.506,392.031,-86.527,-176.164,9.937,148.944
C00699=1142.501,392.278,-86.564,-176.166,9.939,148.945
C00700=1142.497,392.525,-86.601,-176.166,9.941,148.945
C00701=1142.494,392.773,-86.639,-176.167,9.943,148.946
C00702=1142.490,393.020,-86.676,-176.168,9.945,148.947
C00703=1142.486,393.267,-86.713,-176.168,9.948,148.948
C00704=1142.483,393.514,-86.751,-176.169,9.950,148.949
C00705=1142.479,393.761,-86.787,-176.171,9.952,148.950
C00706=1142.475,394.009,-86.824,-176.172,9.954,148.950
C00707=1142.471,394.255,-86.862,-176.172,9.956,148.951
C00708=1142.467,394.503,-86.899,-176.173,9.959,148.952
C00709=1142.463,394.750,-86.936,-176.174,9.961,148.953
C00710=1142.459,394.997,-86.973,-176.175,9.963,148.954
C00711=1142.456,395.245,-87.011,-176.176,9.965,148.954
C00712=1142.452,395.492,-87.048,-176.177,9.967,148.955
C00713=1142.448,395.739,-87.085,-176.178,9.969,148.956
C00714=1142.445,395.986,-87.122,-176.179,9.971,148.957
C00715=1142.441,396.234,-87.159,-176.180,9.973,148.958
C00716=1142.437,396.480,-87.197,-176.182,9.975,148.959
C00717=1142.433,396.728,-87.234,-176.183,9.978,148.959
C00718=1142.429,396.975,-87.271,-176.184,9.980,148.960
C00719=1142.425,397.222,-87.308,-176.185,9.982,148.961
C00720=1142.421,397.469,-87.345,-176.186,9.984,148.962
C00721=1142.418,397.716,-87.383,-176.187,9.986,148.963
C00722=1142.414,397.964,-87.420,-176.188,9.988,148.964
C00723=1142.410,398.211,-87.457,-176.189,9.990,148.964
C00724=1142.407,398.458,-87.495,-176.190,9.992,148.965
C00725=1142.403,398.705,-87.532,-176.192,9.994,148.966
C00726=1142.399,398.952,-87.569,-176.193,9.996,148.967
C00727=1142.396,399.199,-87.606,-176.194,9.998,148.968
C00728=1142.392,399.446,-87.643,-176.196,10.000,148.969
C00729=1142.388,399.694,-87.680,-176.197,10.002,148.970
C00730=1142.385,399.941,-87.718,-176.198,10.004,148.970
C00731=1142.381,400.188,-87.754,-176.199,10.006,148.971
C00732=1142.376,400.435,-87.791,-176.200,10.008,148.972
C00733=1142.373,400.683,-87.829,-176.201,10.010,148.973
C00734=1142.369,400.930,-87.866,-176.202,10.012,148.974
C00735=1142.365,401.177,-87.903,-176.204,10.013,148.974
C00736=1142.361,401.424,-87.941,-176.205,10.015,148.975
C00737=1142.358,401.671,-87.978,-176.206,10.017,148.976
C00738=1142.354,401.919,-88.015,-176.207,10.020,148.977
C00739=1142.350,402.165,-88.052,-176.209,10.022,148.978
C00740=1142.346,402.413,-88.089,-176.210,10.024,148.979
C00741=1142.343,402.660,-88.127,-176.211,10.025,148.980
C00742=1142.339,402.907,-88.164,-176.212,10.027,148.980
C00743=1142.335,403.155,-88.201,-176.214,10.029,148.981
C00744=1142.331,403.401,-88.239,-176.215,10.031,148.982
C00745=1142.327,403.649,-88.276,-176.216,10.033,148.983
C00746=1142.324,403.896,-88.313,-176.217,10.036,148.984
C00747=1142.320,404.143,-88.350,-176.218,10.038,148.985
C00748=1142.316,404.390,-88.387,-176.220,10.039,148.985
C00749=1142.312,404.637,-88.424,-176.221,10.041,148.986
C00750=1142.309,404.885,-88.462,-176.222,10.043,148.987
C00751=1142.304,405.132,-88.499,-176.223,10.045,148.988
C00752=1142.300,405.379,-88.536,-176.224,10.047,148.989
C00753=1142.297,405.626,-88.574,-176.225,10.049,148.990
C00754=1142.293,405.873,-88.610,-176.226,10.051,148.990
C00755=1142.289,406.121,-88.647,-176.227,10.053,148.991
C00756=1142.286,406.368,-88.685,-176.229,10.055,148.992
C00757=1142.282,406.615,-88.722,-176.230,10.057,148.993
C00758=1142.278,406.862,-88.759,-176.231,10.059,148.994
C00759=1142.274,407.110,-88.797,-176.232,10.061,148.994
C00760=1142.270,407.357,-88.834,-176.233,10.063,148.995
C00761=1142.266,407.604,-88.871,-176.234,10.065,148.996
C00762=1142.263,407.851,-88.909,-176.235,10.067,148.997
C00763=1142.259,408.098,-88.945,-176.236,10.069,148.998
C00764=1142.255,408.345,-88.983,-176.237,10.071,148.998
C00765=1142.251,408.592,-89.020,-176.238,10.073,148.999
C00766=1142.248,408.840,-89.057,-176.239,10.075,149.000
C00767=1142.244,409.087,-89.095,-176.240,10.077,149.001
C00768=1142.240,409.334,-89.132,-176.241,10.079,149.002
C00769=1142.236,409.582,-89.169,-176.242,10.081,149.003
C00770=1142.232,409.828,-89.206,-176.243,10.083,149.003
C00771=1142.228,410.075,-89.243,-176.244,10.085,149.004
C00772=1142.225,410.323,-89.280,-176.245,10.087,149.005
C00773=1142.221,410.570,-89.318,-176.246,10.089,149.006
C00774=1142.217,410.817,-89.355,-176.247,10.091,149.007
C00775=1142.213,411.065,-89.392,-176.248,10.093,149.007
C00776=1142.210,411.312,-89.430,-176.249,10.095,149.008
C00777=1142.206,411.559,-89.467,-176.250,10.097,149.009
C00778=1142.201,411.806,-89.503,-176.251,10.100,149.010
C00779=1142.198,412.053,-89.541,-176.252,10.102,149.011
C00780=1142.194,412.300,-89.578,-176.253,10.104,149.011
C00781=1142.190,412.548,-89.615,-176.254,10.106,149.012
C00782=1142.187,412.795,-89.653,-176.255,10.108,149.013
C00783=1142.183,413.042,-89.690,-176.255,10.110,149.013
C00784=1142.179,413.289,-89.727,-176.256,10.112,149.014
C00785=1142.176,413.537,-89.765,-176.257,10.115,149.015
C00786=1142.171,413.784,-89.801,-176.258,10.116,149.016
C00787=1142.168,414.030,-89.839,-176.259,10.118,149.017
C00788=1142.164,414.278,-89.876,-176.260,10.120,149.017
C00789=1142.160,414.525,-89.913,-176.260,10.122,149.018
C00790=1142.158,414.772,-89.950,-176.261,10.125,149.019
C00791=1142.155,415.019,-89.988,-176.262,10.127,149.020
C00792=1142.153,415.267,-90.024,-176.263,10.129,149.020
C00793=1142.152,415.514,-90.061,-176.264,10.131,149.021
C00794=1142.151,415.761,-90.098,-176.264,10.133,149.022
C00795=1142.152,416.008,-90.135,-176.265,10.136,149.023
C00796=1142.152,416.255,-90.172,-176.265,10.137,149.023
C00797=1142.154,416.516,-90.210,-176.267,10.139,149.024
C00798=1142.157,416.777,-90.249,-176.267,10.141,149.025
C00799=1142.160,417.038,-90.287,-176.268,10.144,149.026
C00800=1142.164,417.298,-90.325,-176.268,10.146,149.026
C00801=1141.743,417.302,-90.376,-176.270,10.157,149.030
C00802=1141.740,417.037,-90.337,-176.270,10.154,149.029
C00803=1141.736,416.773,-90.298,-176.269,10.153,149.028
C00804=1141.734,416.509,-90.259,-176.268,10.151,149.028
C00805=1141.732,416.243,-90.220,-176.268,10.148,149.027
C00806=1141.731,415.996,-90.183,-176.267,10.146,149.026
C00807=1141.731,415.750,-90.147,-176.266,10.144,149.025
C00808=1141.731,415.502,-90.110,-176.265,10.142,149.025
C00809=1141.733,415.255,-90.073,-176.264,10.140,149.024
C00810=1141.734,415.008,-90.036,-176.264,10.137,149.023
C00811=1141.737,414.761,-89.998,-176.263,10.135,149.022
C00812=1141.740,414.513,-89.961,-176.262,10.133,149.021
C00813=1141.744,414.266,-89.924,-176.261,10.132,149.021
C00814=1141.748,414.019,-89.887,-176.260,10.130,149.020
C00815=1141.751,413.771,-89.849,-176.260,10.127,149.019
C00816=1141.755,413.525,-89.812,-176.259,10.125,149.018
C00817=1141.759,413.277,-89.775,-176.258,10.123,149.018
C00818=1141.763,413.030,-89.738,-176.257,10.121,149.017
C00819=1141.767,412.783,-89.700,-176.256,10.119,149.016
C00820=1141.771,412.536,-89.663,-176.256,10.116,149.015
C00821=1141.775,412.289,-89.626,-176.255,10.114,149.014
C00822=1141.778,412.041,-89.589,-176.254,10.112,149.014
C00823=1141.782,411.794,-89.552,-176.252,10.110,149.013
C00824=1141.786,411.548,-89.514,-176.252,10.108,149.012
C00825=1141.789,411.300,-89.477,-176.251,10.106,149.011
C00826=1141.793,411.052,-89.440,-176.250,10.104,149.010
C00827=1141.797,410.806,-89.402,-176.249,10.102,149.010
C00828=1141.801,410.558,-89.365,-176.248,10.100,149.009
C00829=1141.805,410.311,-89.328,-176.247,10.098,149.008
C00830=1141.809,410.064,-89.291,-176.246,10.096,149.007
C00831=1141.812,409.816,-89.254,-176.245,10.093,149.006
C00832=1141.816,409.570,-89.216,-176.244,10.091,149.006
C00833=1141.820,409.323,-89.179,-176.243,10.089,149.005
C00834=1141.823,409.075,-89.142,-176.242,10.087,149.004
C00835=1141.827,408.828,-89.104,-176.241,10.085,149.003
C00836=1141.831,408.581,-89.067,-176.240,10.083,149.002
C00837=1141.835,408.334,-89.031,-176.239,10.081,149.002
C00838=1141.839,408.086,-88.993,-176.238,10.079,149.001
C00839=1141.843,407.839,-88.956,-176.236,10.078,149.000
C00840=1141.847,407.592,-88.919,-176.235,10.076,148.999
C00841=1141.850,407.345,-88.881,-176.234,10.074,148.998
C00842=1141.853,407.098,-88.845,-176.233,10.072,148.998
C00843=1141.857,406.851,-88.807,-176.232,10.070,148.997
C00844=1141.861,406.603,-88.770,-176.231,10.068,148.996
C00845=1141.865,406.356,-88.733,-176.230,10.065,148.995
C00846=1141.869,406.110,-88.696,-176.229,10.063,148.994
C00847=1141.872,405.862,-88.658,-176.228,10.061,148.993
C00848=1141.876,405.615,-88.621,-176.227,10.059,148.993
C00849=1141.880,405.368,-88.584,-176.226,10.057,148.992
C00850=1141.883,405.120,-88.547,-176.225,10.055,148.991
C00851=1141.888,404.873,-88.510,-176.223,10.054,148.990
C00852=1141.891,404.626,-88.472,-176.222,10.052,148.989
C00853=1141.895,404.379,-88.435,-176.221,10.050,148.989
C00854=1141.899,404.132,-88.397,-176.220,10.048,148.988
C00855=1141.903,403.885,-88.361,-176.219,10.046,148.987
C00856=1141.907,403.638,-88.324,-176.217,10.044,148.986
C00857=1141.910,403.390,-88.286,-176.216,10.041,148.985
C00858=1141.914,403.143,-88.249,-176.214,10.040,148.984
C00859=1141.918,402.896,-88.212,-176.213,10.038,148.983
C00860=1141.921,402.649,-88.174,-176.212,10.036,148.983
C00861=1141.925,402.401,-88.137,-176.211,10.034,148.982
C00862=1141.930,402.154,-88.100,-176.210,10.032,148.981
C00863=1141.933,401.907,-88.062,-176.209,10.030,148.980
C00864=1141.937,401.660,-88.026,-176.207,10.028,148.979
C00865=1141.941,401.413,-87.988,-176.206,10.026,148.978
C00866=1141.944,401.165,-87.951,-176.205,10.024,148.978
C00867=1141.948,400.918,-87.914,-176.204,10.022,148.977
C00868=1141.952,400.672,-87.876,-176.203,10.020,148.976
C00869=1141.955,400.424,-87.839,-176.201,10.018,148.975
C00870=1141.960,400.176,-87.802,-176.200,10.016,148.974
C00871=1141.963,399.930,-87.765,-176.199,10.014,148.973
C00872=1141.967,399.682,-87.727,-176.197,10.012,148.973
C00873=1141.971,399.435,-87.691,-176.196,10.010,148.972
C00874=1141.975,399.188,-87.653,-176.195,10.008,148.971
C00875=1141.978,398.940,-87.616,-176.194,10.006,148.970
C00876=1141.982,398.694,-87.578,-176.193,10.004,148.969
C00877=1141.986,398.447,-87.541,-176.192,10.002,148.968
C00878=1141.990,398.199,-87.505,-176.191,10.000,148.968
C00879=1141.993,397.952,-87.467,-176.190,9.998,148.967
C00880=1141.997,397.705,-87.430,-176.188,9.997,148.966
C00881=1142.002,397.458,-87.393,-176.187,9.995,148.965
C00882=1142.005,397.211,-87.355,-176.186,9.993,148.964
C00883=1142.009,396.963,-87.318,-176.184,9.990,148.963
C00884=1142.013,396.716,-87.281,-176.183,9.988,148.962
C00885=1142.016,396.469,-87.243,-176.182,9.986,148.962
C00886=1142.020,396.222,-87.206,-176.181,9.984,148.961
C00887=1142.024,395.975,-87.169,-176.180,9.982,148.960
C00888=1142.028,395.727,-87.132,-176.179,9.980,148.959
C00889=1142.032,395.480,-87.095,-176.178,9.978,148.958
C00890=1142.035,395.233,-87.057,-176.178,9.975,148.958
C00891=1142.039,394.986,-87.020,-176.177,9.973,148.957
C00892=1142.043,394.738,-86.983,-176.176,9.971,148.956
C00893=1142.047,394.492,-86.946,-176.175,9.969,148.955
C00894=1142.051,394.245,-86.909,-176.173,9.967,148.954
C00895=1142.054,393.997,-86.871,-176.172,9.965,148.953
C00896=1142.058,393.750,-86.834,-176.171,9.963,148.953
C00897=1142.062,393.503,-86.797,-176.171,9.960,148.952
C00898=1142.066,393.255,-86.760,-176.170,9.958,148.951
C00899=1142.070,393.008,-86.722,-176.169,9.956,148.950
C00900=1142.074,392.761,-86.685,-176.168,9.953,148.949
C00901=1142.077,392.514,-86.647,-176.167,9.951,148.948
C00902=1142.081,392.267,-86.611,-176.166,9.949,148.948
C00903=1142.085,392.020,-86.574,-176.166,9.946,148.947
C00904=1142.088,391.772,-86.536,-176.165,9.945,148.946
C00905=1142.092,391.525,-86.499,-176.165,9.942,148.945
C00906=1142.096,391.238,-86.456,-176.164,9.940,148.944
C00907=1142.101,390.951,-86.413,-176.163,9.937,148.943
C00908=1142.105,390.664,-86.370,-176.162,9.934,148.942
C00909=1142.110,390.377,-86.327,-176.162,9.931,148.941
C00910=1142.113,390.129,-86.289,-176.161,9.929,148.941
C00911=1142.117,389.882,-86.252,-176.160,9.926,148.940
C00912=1142.121,389.635,-86.215,-176.160,9.924,148.939
C00913=1142.124,389.388,-86.177,-176.160,9.921,148.938
C00914=1142.129,389.141,-86.140,-176.160,9.918,148.938
C00915=1142.133,388.893,-86.104,-176.159,9.916,148.937
C00916=1142.136,388.646,-86.066,-176.159,9.913,148.936
C00917=1142.140,388.399,-86.029,-176.158,9.911,148.935
C00918=1142.144,388.152,-85.992,-176.158,9.908,148.935
C00919=1142.148,387.905,-85.954,-176.158,9.905,148.934
C00920=1142.151,387.658,-85.918,-176.158,9.902,148.933
C00921=1142.155,387.410,-85.881,-176.158,9.900,148.932
C00922=1142.159,387.163,-85.844,-176.158,9.897,148.932
C00923=1142.162,386.916,-85.806,-176.158,9.894,148.931
C00924=1142.166,386.669,-85.769,-176.159,9.891,148.930
C00925=1142.170,386.422,-85.732,-176.159,9.888,148.930
C00926=1142.173,386.174,-85.694,-176.159,9.885,148.929
C00927=1142.177,385.927,-85.658,-176.159,9.883,148.928
C00928=1142.181,385.680,-85.621,-176.159,9.879,148.927
C00929=1142.186,385.433,-85.584,-176.160,9.877,148.927
C00930=1142.189,385.185,-85.546,-176.160,9.874,148.926
C00931=1142.193,384.938,-85.509,-176.161,9.870,148.925
C00932=1142.196,384.691,-85.473,-176.161,9.867,148.925
C00933=1142.200,384.444,-85.436,-176.162,9.864,148.924
C00934=1142.204,384.196,-85.399,-176.163,9.860,148.923
C00935=1142.208,383.950,-85.361,-176.164,9.857,148.923
C00936=1142.212,383.703,-85.324,-176.164,9.854,148.922
C00937=1142.215,383.455,-85.287,-176.165,9.851,148.921
C00938=1142.219,383.207,-85.250,-176.166,9.848,148.921
C00939=1142.223,382.960,-85.213,-176.167,9.844,148.920
C00940=1142.227,382.713,-85.177,-176.168,9.841,148.920
C00941=1142.231,382.467,-85.139,-176.169,9.837,148.919
C00942=1142.234,382.219,-85.102,-176.170,9.834,148.918
C00943=1142.238,381.972,-85.065,-176.172,9.830,148.918
C00944=1142.242,381.725,-85.029,-176.173,9.827,148.917
C00945=1142.246,381.477,-84.992,-176.174,9.823,148.917
C00946=1142.249,381.230,-84.955,-176.176,9.819,148.916
C00947=1142.253,380.983,-84.918,-176.178,9.815,148.916
C00948=1142.257,380.735,-84.881,-176.179,9.811,148.915
C00949=1142.261,380.488,-84.844,-176.181,9.808,148.914
C00950=1142.265,380.241,-84.808,-176.182,9.804,148.914
C00951=1142.268,379.993,-84.771,-176.184,9.800,148.913
C00952=1142.272,379.746,-84.734,-176.186,9.796,148.913
C00953=1142.276,379.499,-84.697,-176.187,9.792,148.912
C00954=1142.280,379.252,-84.660,-176.189,9.789,148.912
C00955=1142.284,379.005,-84.624,-176.191,9.785,148.911
C00956=1142.287,378.757,-84.587,-176.192,9.781,148.911
C00957=1142.291,378.510,-84.550,-176.195,9.777,148.910
C00958=1142.296,378.263,-84.513,-176.197,9.773,148.910
C00959=1142.299,378.016,-84.477,-176.198,9.769,148.909
C00960=1142.303,377.769,-84.440,-176.201,9.765,148.908
C00961=1142.307,377.521,-84.403,-176.202,9.761,148.908
C00962=1142.311,377.274,-84.366,-176.205,9.757,148.908
C00963=1142.314,377.027,-84.330,-176.207,9.753,148.907
C00964=1142.318,376.779,-84.294,-176.209,9.749,148.906
C00965=1142.322,376.532,-84.257,-176.211,9.745,148.906
C00966=1142.326,376.285,-84.220,-176.213,9.741,148.906
C00967=1142.330,376.038,-84.184,-176.215,9.737,148.905
C00968=1142.334,375.790,-84.147,-176.218,9.733,148.905
C00969=1142.337,375.544,-84.110,-176.220,9.728,148.904
C00970=1142.341,375.295,-84.074,-176.222,9.725,148.904
C00971=1142.344,375.048,-84.038,-176.225,9.720,148.903
C00972=1142.349,374.801,-84.001,-176.227,9.716,148.903
C00973=1142.353,374.554,-83.964,-176.229,9.712,148.902
C00974=1142.356,374.306,-83.928,-176.232,9.708,148.902
C00975=1142.360,374.059,-83.892,-176.234,9.704,148.902
C00976=1142.364,373.812,-83.855,-176.237,9.699,148.901
C00977=1142.368,373.564,-83.819,-176.239,9.695,148.901
C00978=1142.372,373.317,-83.782,-176.241,9.691,148.900
C00979=1142.376,373.070,-83.746,-176.244,9.687,148.900
C00980=1142.380,372.822,-83.710,-176.246,9.683,148.899
C00981=1142.383,372.576,-83.674,-176.249,9.678,148.899
C00982=1142.388,372.328,-83.637,-176.252,9.674,148.899
C00983=1142.391,372.081,-83.601,-176.254,9.670,148.898
C00984=1142.395,371.833,-83.564,-176.257,9.665,148.898
C00985=1142.398,371.585,-83.528,-176.259,9.662,148.897
C00986=1142.402,371.338,-83.492,-176.262,9.658,148.897
C00987=1142.406,371.091,-83.456,-176.264,9.653,148.896
C00988=1142.410,370.844,-83.419,-176.267,9.649,148.896
C00989=1142.414,370.596,-83.384,-176.269,9.644,148.896
C00990=1142.417,370.349,-83.347,-176.272,9.640,148.895
C00991=1142.422,370.101,-83.311,-176.274,9.636,148.895
C00992=1142.425,369.854,-83.276,-176.277,9.632,148.894
C00993=1142.429,369.607,-83.239,-176.280,9.628,148.894
C00994=1142.434,369.360,-83.204,-176.282,9.623,148.894
C00995=1142.437,369.113,-83.167,-176.285,9.619,148.893
C00996=1142.441,368.865,-83.131,-176.288,9.615,148.893
C00997=1142.445,368.618,-83.096,-176.290,9.610,148.892
C00998=1142.449,368.371,-83.059,-176.293,9.606,148.892
C00999=1142.453,368.123,-83.023,-176.296,9.602,148.892
C01000=1142.456,367.876,-82.988,-176.298,9.597,148.891
C01001=1142.460,367.628,-82.951,-176.301,9.593,148.891
C01002=1142.464,367.381,-82.915,-176.304,9.589,148.890
C01003=1142.468,367.133,-82.880,-176.306,9.585,148.890
C01004=1142.472,366.886,-82.844,-176.309,9.581,148.890
C01005=1142.476,366.639,-82.807,-176.311,9.577,148.889
C01006=1142.479,366.391,-82.772,-176.314,9.573,148.889
C01007=1142.484,366.143,-82.736,-176.317,9.569,148.889
C01008=1142.488,365.897,-82.701,-176.319,9.564,148.888
C01009=1142.492,365.649,-82.665,-176.322,9.560,148.888
C01010=1142.495,365.365,-82.624,-176.325,9.555,148.887
C01011=1142.501,365.081,-82.582,-176.328,9.550,148.887
C01012=1142.505,364.798,-82.542,-176.331,9.546,148.887
C01013=1142.509,364.515,-82.501,-176.334,9.540,148.886
C01014=1142.513,364.267,-82.465,-176.337,9.536,148.886
C01015=1142.517,364.020,-82.430,-176.339,9.533,148.885
C01016=1142.520,363.772,-82.394,-176.342,9.528,148.885
C01017=1142.525,363.524,-82.358,-176.344,9.524,148.885
C01018=1142.528,363.277,-82.323,-176.347,9.520,148.884
C01019=1142.533,363.030,-82.287,-176.350,9.516,148.884
C01020=1142.536,362.782,-82.252,-176.352,9.511,148.883
C01021=1142.540,362.535,-82.216,-176.355,9.507,148.883
C01022=1142.544,362.287,-82.181,-176.357,9.504,148.883
C01023=1142.547,362.040,-82.145,-176.360,9.499,148.882
C01024=1142.552,361.793,-82.110,-176.363,9.495,148.882
C01025=1142.556,361.545,-82.074,-176.365,9.491,148.882
C01026=1142.560,361.298,-82.038,-176.368,9.487,148.881
C01027=1142.563,361.050,-82.003,-176.371,9.482,148.881
C01028=1142.567,360.803,-81.967,-176.373,9.479,148.880
C01029=1142.572,360.555,-81.933,-176.375,9.475,148.880
C01030=1142.575,360.308,-81.897,-176.378,9.470,148.880
C01031=1142.579,360.060,-81.862,-176.381,9.466,148.879
C01032=1142.583,359.813,-81.826,-176.383,9.463,148.879
C01033=1142.587,359.566,-81.791,-176.386,9.459,148.879
C01034=1142.591,359.318,-81.756,-176.388,9.454,148.878
C01035=1142.594,359.070,-81.721,-176.391,9.450,148.878
C01036=1142.598,358.823,-81.685,-176.393,9.447,148.878
C01037=1142.602,358.576,-81.650,-176.396,9.442,148.877
C01038=1142.606,358.328,-81.615,-176.399,9.438,148.877
C01039=1142.610,358.081,-81.579,-176.401,9.434,148.876
C01040=1142.614,357.834,-81.544,-176.403,9.431,148.876
C01041=1142.618,357.586,-81.509,-176.406,9.426,148.876
C01042=1142.622,357.338,-81.474,-176.408,9.422,148.875
C01043=1142.626,357.091,-81.438,-176.411,9.418,148.875
C01044=1142.630,356.843,-81.404,-176.413,9.414,148.875
C01045=1142.634,356.596,-81.368,-176.416,9.410,148.874
C01046=1142.637,356.348,-81.334,-176.419,9.406,148.874
C01047=1142.641,356.101,-81.299,-176.421,9.402,148.874
C01048=1142.645,355.854,-81.263,-176.423,9.398,148.873
C01049=1142.649,355.605,-81.228,-176.426,9.394,148.873
C01050=1142.653,355.359,-81.193,-176.428,9.390,148.873
C01051=1142.657,355.111,-81.158,-176.431,9.386,148.872
C01052=1142.661,354.863,-81.123,-176.434,9.382,148.872
C01053=1142.665,354.616,-81.088,-176.436,9.378,148.871
C01054=1142.668,354.368,-81.054,-176.439,9.374,148.871
C01055=1142.673,354.121,-81.019,-176.441,9.370,148.871
C01056=1142.677,353.873,-80.984,-176.444,9.366,148.871
C01057=1142.681,353.625,-80.949,-176.446,9.362,148.870
C01058=1142.685,353.378,-80.914,-176.449,9.358,148.870
C01059=1142.688,353.131,-80.879,-176.451,9.354,148.869
C01060=1142.693,352.883,-80.845,-176.454,9.350,148.869
C01061=1142.697,352.635,-80.810,-176.456,9.346,148.869
C01062=1142.700,352.388,-80.774,-176.459,9.342,148.869
C01063=1142.704,352.141,-80.741,-176.461,9.338,148.868
C01064=1142.708,351.893,-80.706,-176.464,9.334,148.868
C01065=1142.712,351.646,-80.671,-176.466,9.330,148.867
C01066=1142.716,351.398,-80.636,-176.469,9.327,148.867
C01067=1142.720,351.151,-80.602,-176.471,9.322,148.867
C01068=1142.724,350.902,-80.567,-176.474,9.318,148.867
C01069=1142.728,350.656,-80.532,-176.476,9.315,148.866
C01070=1142.732,350.407,-80.497,-176.479,9.311,148.866
C01071=1142.736,350.160,-80.463,-176.482,9.306,148.865
C01072=1142.740,349.912,-80.428,-176.484,9.303,148.865
C01073=1142.745,349.665,-80.394,-176.486,9.299,148.865
C01074=1142.748,349.418,-80.359,-176.489,9.294,148.864
C01075=1142.752,349.170,-80.324,-176.491,9.291,148.864
C01076=1142.756,348.922,-80.290,-176.494,9.287,148.864
C01077=1142.760,348.675,-80.256,-176.496,9.284,148.864
C01078=1142.764,348.427,-80.221,-176.499,9.279,148.863
C01079=1142.768,348.180,-80.187,-176.502,9.275,148.863
C01080=1142.772,347.932,-80.152,-176.504,9.272,148.863
C01081=1142.776,347.684,-80.118,-176.507,9.267,148.862
C01082=1142.780,347.436,-80.083,-176.509,9.263,148.862
C01083=1142.784,347.189,-80.049,-176.512,9.260,148.862
C01084=1142.787,346.941,-80.015,-176.515,9.256,148.861
C01085=1142.792,346.694,-79.980,-176.517,9.251,148.861
C01086=1142.795,346.446,-79.946,-176.519,9.248,148.861
C01087=1142.800,346.199,-79.912,-176.522,9.244,148.860
C01088=1142.804,345.951,-79.877,-176.524,9.240,148.860
C01089=1142.807,345.703,-79.843,-176.527,9.236,148.860
C01090=1142.812,345.456,-79.808,-176.530,9.232,148.859
C01091=1142.815,345.208,-79.774,-176.532,9.229,148.859
C01092=1142.820,344.961,-79.740,-176.534,9.224,148.859
C01093=1142.824,344.714,-79.706,-176.537,9.220,148.858
C01094=1142.828,344.465,-79.671,-176.540,9.217,148.858
C01095=1142.832,344.218,-79.638,-176.542,9.213,148.858
C01096=1142.836,343.970,-79.603,-176.545,9.209,148.858
C01097=1142.840,343.722,-79.569,-176.547,9.205,148.857
C01098=1142.843,343.475,-79.535,-176.550,9.201,148.857
C01099=1142.847,343.227,-79.500,-176.552,9.198,148.857
C01100=1142.852,342.979,-79.467,-176.555,9.193,148.856
C01101=1142.856,342.732,-79.433,-176.557,9.190,148.856
C01102=1142.859,342.484,-79.399,-176.560,9.186,148.856
C01103=1142.864,342.237,-79.364,-176.563,9.181,148.855
C01104=1142.868,341.989,-79.331,-176.565,9.178,148.855
C01105=1142.871,341.741,-79.297,-176.568,9.174,148.855
C01106=1142.876,341.494,-79.262,-176.570,9.171,148.855
C01107=1142.880,341.246,-79.229,-176.573,9.166,148.854
C01108=1142.883,340.998,-79.195,-176.576,9.162,148.854
C01109=1142.888,340.751,-79.160,-176.577,9.159,148.854
C01110=1142.892,340.503,-79.127,-176.580,9.155,148.853
C01111=1142.895,340.255,-79.093,-176.583,9.151,148.853
C01112=1142.900,340.007,-79.059,-176.585,9.147,148.853
C01113=1142.904,339.760,-79.025,-176.588,9.143,148.852
C01114=1142.909,339.480,-78.987,-176.591,9.139,148.852
C01115=1142.913,339.199,-78.948,-176.594,9.134,148.852
C01116=1142.917,338.919,-78.910,-176.596,9.130,148.852
C01117=1142.922,338.638,-78.872,-176.599,9.126,148.851
C01118=1142.926,338.390,-78.839,-176.602,9.122,148.851
C01119=1142.929,338.143,-78.805,-176.604,9.119,148.851
C01120=1142.934,337.895,-78.771,-176.607,9.115,148.850
C01121=1142.938,337.647,-78.737,-176.610,9.111,148.850
C01122=1142.942,337.400,-78.704,-176.612,9.107,148.850
C01123=1142.946,337.152,-78.670,-176.615,9.103,148.850
C01124=1142.950,336.904,-78.636,-176.617,9.100,148.849
C01125=1142.955,336.656,-78.603,-176.620,9.096,148.849
C01126=1142.958,336.409,-78.569,-176.622,9.092,148.849
C01127=1142.963,336.161,-78.536,-176.625,9.088,148.848
C01128=1142.966,335.913,-78.501,-176.628,9.084,148.848
C01129=1142.970,335.666,-78.468,-176.630,9.081,148.848
C01130=1142.974,335.418,-78.435,-176.633,9.076,148.848
C01131=1142.979,335.171,-78.401,-176.635,9.073,148.847
C01132=1142.983,334.923,-78.367,-176.638,9.069,148.847
C01133=1142.986,334.674,-78.334,-176.640,9.066,148.847
C01134=1142.990,334.427,-78.301,-176.643,9.061,148.846
C01135=1142.994,334.180,-78.267,-176.645,9.058,148.846
C01136=1142.998,333.932,-78.234,-176.648,9.054,148.846
C01137=1143.003,333.684,-78.201,-176.650,9.051,148.846
C01138=1143.007,333.436,-78.167,-176.653,9.046,148.846
C01139=1143.010,333.188,-78.134,-176.656,9.042,148.845
C01140=1143.014,332.941,-78.100,-176.658,9.039,148.845
C01141=1143.018,332.693,-78.067,-176.661,9.035,148.845
C01142=1143.022,332.445,-78.034,-176.663,9.031,148.845
C01143=1143.026,332.198,-78.001,-176.666,9.027,148.844
C01144=1143.031,331.950,-77.967,-176.668,9.024,148.844
C01145=1143.035,331.702,-77.934,-176.671,9.020,148.844
C01146=1143.039,331.454,-77.901,-176.673,9.016,148.843
C01147=1143.043,331.207,-77.868,-176.676,9.012,148.843
C01148=1143.047,330.958,-77.834,-176.679,9.009,148.843
C01149=1143.050,330.711,-77.801,-176.682,9.005,148.843
C01150=1143.054,330.463,-77.767,-176.684,9.002,148.843
C01151=1143.059,330.216,-77.734,-176.686,8.997,148.842
C01152=1143.063,329.968,-77.701,-176.689,8.994,148.842
C01153=1143.067,329.720,-77.668,-176.692,8.990,148.842
C01154=1143.071,329.473,-77.635,-176.694,8.987,148.842
C01155=1143.075,329.224,-77.602,-176.697,8.983,148.841
C01156=1143.080,328.976,-77.569,-176.699,8.979,148.841
C01157=1143.084,328.729,-77.536,-176.702,8.975,148.841
C01158=1143.088,328.481,-77.503,-176.704,8.972,148.841
C01159=1143.092,328.233,-77.470,-176.707,8.968,148.840
C01160=1143.095,327.986,-77.437,-176.709,8.964,148.840
C01161=1143.100,327.738,-77.404,-176.712,8.960,148.840
C01162=1143.104,327.490,-77.371,-176.715,8.957,148.840
C01163=1143.108,327.243,-77.338,-176.718,8.953,148.839
C01164=1143.112,326.994,-77.305,-176.720,8.950,148.839
C01165=1143.116,326.747,-77.272,-176.723,8.946,148.839
C01166=1143.120,326.499,-77.240,-176.725,8.942,148.839
C01167=1143.124,326.251,-77.206,-176.728,8.938,148.839
C01168=1143.128,326.004,-77.173,-176.730,8.935,148.838
C01169=1143.133,325.755,-77.141,-176.733,8.931,148.838
C01170=1143.137,325.508,-77.108,-176.735,8.927,148.838
C01171=1143.140,325.260,-77.075,-176.738,8.923,148.838
C01172=1143.145,325.012,-77.043,-176.741,8.920,148.837
C01173=1143.149,324.764,-77.009,-176.743,8.916,148.837
C01174=1143.153,324.516,-76.976,-176.746,8.913,148.837
C01175=1143.157,324.268,-76.944,-176.749,8.909,148.837
C01176=1143.161,324.021,-76.911,-176.751,8.905,148.836
C01177=1143.165,323.773,-76.878,-176.754,8.901,148.836
C01178=1143.169,323.525,-76.846,-176.756,8.898,148.836
C01179=1143.173,323.277,-76.813,-176.759,8.894,148.836
C01180=1143.177,323.029,-76.780,-176.762,8.891,148.836
C01181=1143.180,322.781,-76.748,-176.764,8.887,148.835
C01182=1143.185,322.534,-76.715,-176.767,8.883,148.835
C01183=1143.190,322.286,-76.683,-176.770,8.879,148.835
C01184=1143.193,322.039,-76.650,-176.772,8.876,148.835
C01185=1143.198,321.790,-76.618,-176.774,8.873,148.835
C01186=1143.202,321.543,-76.585,-176.777,8.869,148.834
C01187=1143.205,321.294,-76.553,-176.780,8.865,148.834
C01188=1143.209,321.047,-76.520,-176.783,8.861,148.834
C01189=1143.213,320.799,-76.488,-176.785,8.858,148.834
C01190=1143.217,320.551,-76.455,-176.788,8.854,148.834
C01191=1143.221,320.303,-76.423,-176.790,8.851,148.833
C01192=1143.226,320.055,-76.391,-176.793,8.847,148.833
C01193=1143.230,319.808,-76.358,-176.795,8.843,148.833
C01194=1143.234,319.560,-76.326,-176.798,8.839,148.833
C01195=1143.238,319.312,-76.293,-176.801,8.836,148.833
C01196=1143.242,319.064,-76.261,-176.803,8.833,148.832
C01197=1143.246,318.815,-76.228,-176.806,8.829,148.832
C01198=1143.250,318.569,-76.196,-176.808,8.825,148.832
C01199=1143.255,318.320,-76.164,-176.811,8.821,148.832
C01200=1143.258,318.072,-76.132,-176.814,8.818,148.832
C01201=1143.263,317.825,-76.099,-176.816,8.814,148.831
C01202=1143.266,317.577,-76.067,-176.819,8.811,148.831
C01203=1143.271,317.329,-76.035,-176.821,8.808,148.831
C01204=1143.275,317.081,-76.003,-176.824,8.803,148.831
C01205=1143.279,316.833,-75.970,-176.826,8.800,148.831
C01206=1143.283,316.585,-75.938,-176.829,8.796,148.830
C01207=1143.287,316.337,-75.906,-176.832,8.793,148.830
C01208=1143.292,316.089,-75.874,-176.835,8.789,148.830
C01209=1143.295,315.841,-75.842,-176.837,8.786,148.830
C01210=1143.300,315.593,-75.810,-176.840,8.783,148.830
C01211=1143.303,315.346,-75.777,-176.843,8.778,148.829
C01212=1143.307,315.098,-75.746,-176.845,8.775,148.829
C01213=1143.312,314.850,-75.713,-176.848,8.771,148.829
C01214=1143.316,314.602,-75.681,-176.850,8.768,148.829
C01215=1143.320,314.354,-75.649,-176.852,8.765,148.829
C01216=1143.324,314.106,-75.618,-176.855,8.761,148.828
C01217=1143.328,313.858,-75.586,-176.858,8.758,148.828
C01218=1143.333,313.580,-75.550,-176.861,8.754,148.828
C01219=1143.337,313.303,-75.514,-176.864,8.749,148.828
C01220=1143.342,313.025,-75.478,-176.867,8.745,148.828
C01221=1143.347,312.747,-75.442,-176.870,8.741,148.828
C01222=1143.350,312.499,-75.410,-176.872,8.738,148.827
C01223=1143.354,312.251,-75.378,-176.875,8.734,148.827
C01224=1143.360,312.003,-75.347,-176.878,8.731,148.827
C01225=1143.363,311.755,-75.315,-176.881,8.727,148.827
C01226=1143.367,311.507,-75.283,-176.883,8.724,148.827
C01227=1143.372,311.259,-75.251,-176.885,8.720,148.827
C01228=1143.376,311.011,-75.219,-176.888,8.716,148.826
C01229=1143.380,310.764,-75.188,-176.891,8.713,148.826
C01230=1143.384,310.516,-75.156,-176.893,8.710,148.826
C01231=1143.387,310.268,-75.124,-176.896,8.706,148.826
C01232=1143.393,310.020,-75.093,-176.899,8.703,148.826
C01233=1143.396,309.772,-75.061,-176.902,8.699,148.826
C01234=1143.400,309.524,-75.029,-176.904,8.695,148.825
C01235=1143.404,309.276,-74.998,-176.906,8.692,148.825
C01236=1143.408,309.028,-74.966,-176.910,8.688,148.825
C01237=1143.414,308.780,-74.935,-176.912,8.685,148.825
C01238=1143.417,308.532,-74.903,-176.914,8.682,148.825
C01239=1143.421,308.284,-74.871,-176.917,8.678,148.825
C01240=1143.425,308.036,-74.839,-176.920,8.675,148.824
C01241=1143.429,307.788,-74.808,-176.923,8.671,148.824
C01242=1143.434,307.540,-74.777,-176.925,8.668,148.824
C01243=1143.437,307.292,-74.745,-176.928,8.664,148.824
C01244=1143.443,307.044,-74.714,-176.931,8.660,148.824
C01245=1143.446,306.796,-74.682,-176.933,8.657,148.824
C01246=1143.450,306.547,-74.651,-176.936,8.654,148.824
C01247=1143.455,306.300,-74.619,-176.939,8.650,148.824
C01248=1143.458,306.052,-74.587,-176.941,8.647,148.823
C01249=1143.463,305.804,-74.556,-176.944,8.644,148.823
C01250=1143.467,305.556,-74.525,-176.947,8.640,148.823
C01251=1143.471,305.308,-74.494,-176.949,8.636,148.823
C01252=1143.475,305.060,-74.462,-176.951,8.633,148.823
C01253=1143.480,304.812,-74.431,-176.955,8.629,148.823
C01254=1143.483,304.564,-74.399,-176.957,8.626,148.823
C01255=1143.488,304.316,-74.369,-176.959,8.623,148.822
C01256=1143.492,304.068,-74.337,-176.962,8.619,148.822
C01257=1143.496,303.820,-74.306,-176.965,8.616,148.822
C01258=1143.500,303.572,-74.274,-176.967,8.613,148.822
C01259=1143.505,303.324,-74.243,-176.970,8.608,148.822
C01260=1143.509,303.077,-74.212,-176.973,8.606,148.822
C01261=1143.513,302.828,-74.181,-176.975,8.602,148.822
C01262=1143.518,302.580,-74.150,-176.978,8.598,148.822
C01263=1143.521,302.332,-74.118,-176.981,8.595,148.821
C01264=1143.526,302.084,-74.087,-176.983,8.592,148.821
C01265=1143.530,301.836,-74.056,-176.986,8.588,148.821
C01266=1143.534,301.588,-74.025,-176.989,8.585,148.821
C01267=1143.538,301.340,-73.994,-176.991,8.582,148.821
C01268=1143.542,301.093,-73.963,-176.994,8.578,148.821
C01269=1143.546,300.845,-73.932,-176.997,8.574,148.821
C01270=1143.550,300.596,-73.901,-176.999,8.571,148.821
C01271=1143.555,300.348,-73.870,-177.002,8.567,148.820
C01272=1143.559,300.100,-73.838,-177.005,8.564,148.820
C01273=1143.563,299.852,-73.808,-177.007,8.561,148.820
C01274=1143.568,299.604,-73.777,-177.010,8.557,148.820
C01275=1143.571,299.356,-73.746,-177.013,8.554,148.820
C01276=1143.576,299.108,-73.716,-177.015,8.551,148.820
C01277=1143.580,298.860,-73.684,-177.018,8.547,148.820
C01278=1143.584,298.612,-73.653,-177.021,8.544,148.820
C01279=1143.589,298.364,-73.622,-177.024,8.541,148.820
C01280=1143.592,298.115,-73.592,-177.026,8.537,148.819
C01281=1143.597,297.867,-73.561,-177.029,8.533,148.819
C01282=1143.601,297.619,-73.530,-177.032,8.530,148.819
C01283=1143.605,297.371,-73.499,-177.034,8.527,148.819
C01284=1143.609,297.124,-73.468,-177.037,8.523,148.819
C01285=1143.613,296.876,-73.437,-177.040,8.520,148.819
C01286=1143.617,296.627,-73.406,-177.042,8.517,148.819
C01287=1143.622,296.379,-73.375,-177.045,8.514,148.819
C01288=1143.626,296.132,-73.345,-177.048,8.510,148.819
C01289=1143.630,295.883,-73.314,-177.050,8.507,148.819
C01290=1143.635,295.635,-73.283,-177.053,8.504,148.818
C01291=1143.638,295.387,-73.253,-177.056,8.499,148.818
C01292=1143.642,295.139,-73.222,-177.058,8.497,148.818
C01293=1143.647,294.891,-73.191,-177.061,8.493,148.818
C01294=1143.651,294.643,-73.161,-177.064,8.490,148.818
C01295=1143.656,294.394,-73.131,-177.066,8.486,148.818
C01296=1143.659,294.146,-73.101,-177.069,8.483,148.818
C01297=1143.664,293.898,-73.070,-177.072,8.480,148.818
C01298=1143.668,293.650,-73.039,-177.074,8.476,148.818
C01299=1143.672,293.402,-73.008,-177.077,8.473,148.818
C01300=1143.676,293.154,-72.978,-177.080,8.470,148.817
C01301=1143.680,292.906,-72.948,-177.082,8.467,148.817
C01302=1143.685,292.658,-72.917,-177.085,8.463,148.817
C01303=1143.688,292.409,-72.887,-177.088,8.460,148.817
C01304=1143.693,292.161,-72.856,-177.090,8.457,148.817
C01305=1143.698,291.913,-72.825,-177.093,8.453,148.817
C01306=1143.701,291.666,-72.795,-177.096,8.450,148.817
C01307=1143.706,291.418,-72.764,-177.098,8.446,148.817
C01308=1143.710,291.169,-72.735,-177.101,8.443,148.817
C01309=1143.714,290.921,-72.704,-177.104,8.440,148.817
C01310=1143.718,290.673,-72.674,-177.107,8.436,148.817
C01311=1143.723,290.425,-72.644,-177.109,8.433,148.816
C01312=1143.727,290.177,-72.614,-177.112,8.430,148.817
C01313=1143.731,289.928,-72.582,-177.114,8.427,148.816
C01314=1143.735,289.680,-72.553,-177.118,8.423,148.816
C01315=1143.740,289.432,-72.522,-177.120,8.420,148.816
C01316=1143.744,289.184,-72.492,-177.123,8.417,148.816
C01317=1143.748,288.936,-72.463,-177.125,8.414,148.816
C01318=1143.752,288.688,-72.432,-177.129,8.410,148.816
C01319=1143.756,288.439,-72.402,-177.131,8.407,148.816
C01320=1143.761,288.191,-72.371,-177.134,8.404,148.816
C01321=1143.764,287.944,-72.341,-177.136,8.400,148.816
C01322=1143.769,287.668,-72.308,-177.139,8.397,148.816
C01323=1143.774,287.392,-72.274,-177.142,8.393,148.816
C01324=1143.779,287.117,-72.242,-177.145,8.390,148.816
C01325=1143.783,286.842,-72.208,-177.148,8.386,148.815
C01326=1143.788,286.594,-72.177,-177.151,8.383,148.815
C01327=1143.792,286.345,-72.148,-177.154,8.379,148.815
C01328=1143.796,286.097,-72.118,-177.156,8.376,148.815
C01329=1143.801,285.849,-72.087,-177.159,8.373,148.815
C01330=1143.805,285.601,-72.058,-177.162,8.370,148.815
C01331=1143.809,285.353,-72.028,-177.164,8.367,148.815
C01332=1143.814,285.105,-71.998,-177.167,8.362,148.815
C01333=1143.818,284.856,-71.968,-177.170,8.360,148.815
C01334=1143.821,284.608,-71.938,-177.172,8.356,148.815
C01335=1143.825,284.360,-71.908,-177.175,8.353,148.815
C01336=1143.830,284.112,-71.878,-177.177,8.350,148.815
C01337=1143.834,283.864,-71.848,-177.181,8.346,148.815
C01338=1143.838,283.615,-71.819,-177.184,8.343,148.815
C01339=1143.843,283.367,-71.789,-177.186,8.340,148.815
C01340=1143.847,283.119,-71.758,-177.189,8.337,148.815
C01341=1143.851,282.871,-71.729,-177.191,8.334,148.815
C01342=1143.855,282.623,-71.700,-177.194,8.330,148.815
C01343=1143.859,282.375,-71.669,-177.197,8.327,148.814
C01344=1143.864,282.126,-71.639,-177.200,8.324,148.814
C01345=1143.868,281.878,-71.610,-177.202,8.321,148.814
C01346=1143.873,281.630,-71.580,-177.205,8.318,148.814
C01347=1143.877,281.381,-71.551,-177.208,8.314,148.814
C01348=1143.881,281.133,-71.521,-177.210,8.311,148.814
C01349=1143.885,280.886,-71.491,-177.213,8.308,148.814
C01350=1143.890,280.637,-71.461,-177.216,8.305,148.814
C01351=1143.894,280.389,-71.432,-177.218,8.302,148.814
C01352=1143.898,280.140,-71.402,-177.222,8.298,148.814
C01353=1143.902,279.892,-71.373,-177.224,8.295,148.814
C01354=1143.907,279.645,-71.344,-177.227,8.292,148.814
C01355=1143.911,279.396,-71.314,-177.229,8.289,148.814
C01356=1143.915,279.148,-71.285,-177.232,8.286,148.814
C01357=1143.920,278.900,-71.255,-177.235,8.283,148.814
C01358=1143.924,278.652,-71.226,-177.238,8.279,148.814
C01359=1143.928,278.403,-71.197,-177.240,8.276,148.814
C01360=1143.932,278.155,-71.167,-177.243,8.273,148.814
C01361=1143.936,277.907,-71.138,-177.245,8.269,148.814
C01362=1143.941,277.658,-71.108,-177.248,8.266,148.814
C01363=1143.946,277.410,-71.078,-177.251,8.264,148.814
C01364=1143.950,277.162,-71.049,-177.254,8.259,148.814
C01365=1143.954,276.913,-71.019,-177.257,8.257,148.814
C01366=1143.958,276.665,-70.990,-177.259,8.254,148.814
C01367=1143.962,276.418,-70.961,-177.262,8.250,148.814
C01368=1143.966,276.170,-70.932,-177.265,8.247,148.814
C01369=1143.970,275.921,-70.902,-177.267,8.244,148.814
C01370=1143.975,275.673,-70.873,-177.270,8.240,148.813
C01371=1143.979,275.425,-70.843,-177.273,8.237,148.813
C01372=1143.983,275.176,-70.815,-177.276,8.235,148.814
C01373=1143.987,274.928,-70.785,-177.278,8.231,148.813
C01374=1143.992,274.680,-70.756,-177.281,8.228,148.813
C01375=1143.996,274.432,-70.727,-177.284,8.225,148.813
C01376=1144.001,274.184,-70.697,-177.286,8.222,148.813
C01377=1144.005,273.935,-70.669,-177.289,8.218,148.813
C01378=1144.009,273.686,-70.639,-177.292,8.215,148.813
C01379=1144.013,273.438,-70.610,-177.295,8.213,148.813
C01380=1144.018,273.191,-70.581,-177.297,8.209,148.813
C01381=1144.022,272.942,-70.552,-177.300,8.206,148.813
C01382=1144.026,272.694,-70.523,-177.303,8.203,148.813
C01383=1144.030,272.445,-70.494,-177.305,8.200,148.813
C01384=1144.035,272.197,-70.465,-177.308,8.197,148.813
C01385=1144.040,271.949,-70.436,-177.311,8.193,148.813
C01386=1144.043,271.701,-70.407,-177.314,8.191,148.813
C01387=1144.048,271.452,-70.378,-177.317,8.187,148.813
C01388=1144.052,271.204,-70.349,-177.319,8.184,148.813
C01389=1144.057,270.956,-70.320,-177.322,8.181,148.813
C01390=1144.061,270.707,-70.291,-177.324,8.178,148.813
C01391=1144.064,270.459,-70.262,-177.327,8.175,148.813
C01392=1144.069,270.211,-70.233,-177.330,8.172,148.813
C01393=1144.074,269.963,-70.204,-177.333,8.169,148.813
C01394=1144.078,269.714,-70.175,-177.336,8.165,148.813
C01395=1144.082,269.466,-70.147,-177.338,8.162,148.813
C01396=1144.086,269.217,-70.118,-177.341,8.159,148.813
C01397=1144.091,268.970,-70.089,-177.344,8.157,148.813
C01398=1144.095,268.721,-70.060,-177.346,8.153,148.813
C01399=1144.099,268.473,-70.031,-177.349,8.150,148.813
C01400=1144.104,268.225,-70.003,-177.352,8.147,148.813
C01401=1144.108,267.976,-69.973,-177.355,8.144,148.813
C01402=1144.112,267.728,-69.945,-177.358,8.140,148.813
C01403=1144.116,267.479,-69.916,-177.360,8.137,148.813
C01404=1144.121,267.231,-69.887,-177.363,8.135,148.813
C01405=1144.125,266.983,-69.859,-177.366,8.132,148.813
C01406=1144.129,266.735,-69.830,-177.369,8.129,148.813
C01407=1144.134,266.486,-69.801,-177.371,8.125,148.813
C01408=1144.138,266.238,-69.773,-177.374,8.122,148.813
C01409=1144.143,265.990,-69.744,-177.377,8.120,148.813
C01410=1144.146,265.742,-69.716,-177.379,8.117,148.813
C01411=1144.151,265.493,-69.687,-177.382,8.113,148.813
C01412=1144.156,265.245,-69.659,-177.385,8.110,148.813
C01413=1144.159,264.997,-69.630,-177.388,8.107,148.813
C01414=1144.164,264.748,-69.601,-177.391,8.104,148.813
C01415=1144.168,264.500,-69.573,-177.394,8.101,148.813
C01416=1144.173,264.251,-69.545,-177.396,8.098,148.813
C01417=1144.177,264.004,-69.516,-177.399,8.095,148.813
C01418=1144.181,263.755,-69.488,-177.401,8.092,148.813
C01419=1144.186,263.506,-69.459,-177.404,8.089,148.813
C01420=1144.190,263.258,-69.431,-177.407,8.086,148.814
C01421=1144.195,263.009,-69.402,-177.410,8.083,148.814
C01422=1144.199,262.761,-69.374,-177.412,8.080,148.813
C01423=1144.203,262.513,-69.345,-177.415,8.077,148.814
C01424=1144.208,262.265,-69.317,-177.418,8.074,148.814
C01425=1144.212,262.016,-69.289,-177.420,8.071,148.814
C01426=1144.217,261.743,-69.258,-177.424,8.067,148.814
C01427=1144.221,261.470,-69.227,-177.427,8.064,148.814
C01428=1144.226,261.195,-69.196,-177.430,8.060,148.814
C01429=1144.231,260.923,-69.164,-177.433,8.058,148.814
C01430=1144.236,260.674,-69.136,-177.435,8.054,148.814
C01431=1144.239,260.426,-69.108,-177.438,8.051,148.814
C01432=1144.244,260.178,-69.080,-177.441,8.048,148.814
C01433=1144.248,259.929,-69.051,-177.444,8.045,148.814
C01434=1144.252,259.680,-69.023,-177.447,8.042,148.814
C01435=1144.256,259.433,-68.995,-177.450,8.039,148.814
C01436=1144.261,259.184,-68.966,-177.452,8.036,148.814
C01437=1144.265,258.935,-68.939,-177.455,8.033,148.814
C01438=1144.270,258.686,-68.911,-177.458,8.030,148.814
C01439=1144.274,258.438,-68.883,-177.460,8.027,148.814
C01440=1144.279,258.191,-68.855,-177.463,8.024,148.814
C01441=1144.283,257.942,-68.826,-177.466,8.021,148.814
C01442=1144.287,257.694,-68.799,-177.469,8.018,148.814
C01443=1144.291,257.445,-68.770,-177.471,8.015,148.814
C01444=1144.296,257.197,-68.743,-177.474,8.012,148.814
C01445=1144.300,256.948,-68.715,-177.477,8.009,148.814
C01446=1144.305,256.700,-68.687,-177.479,8.006,148.814
C01447=1144.308,256.451,-68.659,-177.482,8.003,148.814
C01448=1144.314,256.203,-68.630,-177.485,8.000,148.814
C01449=1144.317,255.955,-68.602,-177.488,7.997,148.814
C01450=1144.322,255.706,-68.575,-177.491,7.994,148.815
C01451=1144.326,255.458,-68.547,-177.493,7.991,148.815
C01452=1144.331,255.209,-68.519,-177.496,7.988,148.815
C01453=1144.335,254.961,-68.492,-177.499,7.986,148.815
C01454=1144.339,254.712,-68.463,-177.501,7.982,148.815
C01455=1144.344,254.464,-68.436,-177.504,7.979,148.815
C01456=1144.348,254.216,-68.408,-177.507,7.976,148.815
C01457=1144.353,253.967,-68.380,-177.510,7.973,148.815
C01458=1144.357,253.719,-68.352,-177.512,7.971,148.815
C01459=1144.362,253.471,-68.325,-177.515,7.968,148.815
C01460=1144.365,253.222,-68.297,-177.518,7.965,148.815
C01461=1144.370,252.974,-68.269,-177.521,7.962,148.815
C01462=1144.374,252.725,-68.242,-177.524,7.959,148.815
C01463=1144.378,252.477,-68.214,-177.526,7.956,148.815
C01464=1144.384,252.228,-68.186,-177.529,7.953,148.815
C01465=1144.387,251.980,-68.158,-177.532,7.950,148.815
C01466=1144.392,251.731,-68.131,-177.535,7.947,148.815
C01467=1144.396,251.483,-68.103,-177.538,7.944,148.815
C01468=1144.400,251.235,-68.075,-177.540,7.941,148.816
C01469=1144.405,250.986,-68.048,-177.543,7.938,148.815
C01470=1144.409,250.738,-68.021,-177.545,7.935,148.815
C01471=1144.413,250.489,-67.993,-177.548,7.932,148.816
C01472=1144.418,250.241,-67.966,-177.551,7.929,148.816
C01473=1144.422,249.993,-67.938,-177.554,7.926,148.816
C01474=1144.427,249.744,-67.911,-177.557,7.923,148.816
C01475=1144.431,249.496,-67.883,-177.559,7.921,148.816
C01476=1144.435,249.247,-67.856,-177.562,7.918,148.816
C01477=1144.440,248.999,-67.829,-177.565,7.915,148.816
C01478=1144.444,248.750,-67.801,-177.568,7.912,148.816
C01479=1144.448,248.502,-67.773,-177.571,7.909,148.816
C01480=1144.453,248.254,-67.746,-177.573,7.906,148.816
C01481=1144.457,248.005,-67.719,-177.576,7.903,148.816
C01482=1144.461,247.756,-67.691,-177.579,7.900,148.816
C01483=1144.466,247.508,-67.664,-177.582,7.897,148.816
C01484=1144.470,247.260,-67.636,-177.584,7.894,148.816
C01485=1144.475,247.011,-67.609,-177.587,7.891,148.817
C01486=1144.479,246.762,-67.582,-177.590,7.888,148.817
C01487=1144.483,246.514,-67.554,-177.593,7.885,148.817
C01488=1144.488,246.266,-67.527,-177.596,7.883,148.817
C01489=1144.493,246.017,-67.500,-177.598,7.880,148.817
C01490=1144.497,245.769,-67.473,-177.601,7.877,148.817
C01491=1144.501,245.519,-67.445,-177.604,7.874,148.817
C01492=1144.505,245.272,-67.418,-177.607,7.871,148.817
C01493=1144.510,245.023,-67.391,-177.610,7.868,148.817
C01494=1144.514,244.775,-67.364,-177.612,7.865,148.817
C01495=1144.519,244.526,-67.337,-177.615,7.862,148.817
C01496=1144.523,244.277,-67.310,-177.618,7.859,148.817
C01497=1144.528,244.029,-67.283,-177.620,7.857,148.817
C01498=1144.532,243.781,-67.256,-177.623,7.854,148.818
C01499=1144.536,243.533,-67.228,-177.626,7.851,148.818
C01500=1144.541,243.284,-67.201,-177.629,7.848,148.818
C01501=1144.545,243.036,-67.174,-177.631,7.845,148.818
C01502=1144.550,242.787,-67.147,-177.634,7.842,148.818
C01503=1144.553,242.538,-67.120,-177.637,7.839,148.818
C01504=1144.558,242.290,-67.093,-177.640,7.837,148.818
C01505=1144.563,242.041,-67.066,-177.643,7.834,148.818
C01506=1144.567,241.793,-67.039,-177.645,7.831,148.818
C01507=1144.571,241.545,-67.013,-177.648,7.828,148.818
C01508=1144.576,241.296,-66.986,-177.651,7.825,148.818
C01509=1144.581,241.048,-66.959,-177.654,7.822,148.818
C01510=1144.585,240.799,-66.932,-177.656,7.819,148.818
C01511=1144.589,240.551,-66.905,-177.660,7.816,148.819
C01512=1144.593,240.301,-66.878,-177.662,7.814,148.819
C01513=1144.598,240.053,-66.851,-177.665,7.811,148.819
C01514=1144.602,239.804,-66.825,-177.668,7.809,148.819
C01515=1144.607,239.556,-66.798,-177.670,7.806,148.819
C01516=1144.611,239.307,-66.771,-177.673,7.803,148.819
C01517=1144.615,239.059,-66.744,-177.676,7.800,148.819
C01518=1144.620,238.811,-66.717,-177.679,7.797,148.819
C01519=1144.625,238.562,-66.691,-177.681,7.794,148.819
C01520=1144.629,238.313,-66.664,-177.684,7.791,148.820
C01521=1144.633,238.065,-66.637,-177.687,7.788,148.820
C01522=1144.638,237.817,-66.610,-177.690,7.785,148.820
C01523=1144.642,237.568,-66.584,-177.692,7.783,148.820
C01524=1144.647,237.319,-66.557,-177.695,7.780,148.820
C01525=1144.651,237.071,-66.531,-177.698,7.777,148.820
C01526=1144.656,236.823,-66.504,-177.701,7.775,148.820
C01527=1144.660,236.574,-66.477,-177.704,7.772,148.820
C01528=1144.664,236.325,-66.451,-177.706,7.769,148.820
C01529=1144.669,236.077,-66.424,-177.709,7.766,148.820
C01530=1144.674,235.805,-66.395,-177.712,7.763,148.821
C01531=1144.678,235.533,-66.366,-177.715,7.760,148.821
C01532=1144.683,235.261,-66.337,-177.718,7.756,148.821
C01533=1144.688,234.990,-66.308,-177.721,7.754,148.821
C01534=1144.693,234.741,-66.282,-177.724,7.751,148.821
C01535=1144.697,234.492,-66.255,-177.727,7.748,148.821
C01536=1144.702,234.243,-66.229,-177.730,7.745,148.821
C01537=1144.706,233.995,-66.203,-177.732,7.743,148.821
C01538=1144.710,233.747,-66.175,-177.735,7.740,148.821
C01539=1144.715,233.498,-66.150,-177.738,7.737,148.822
C01540=1144.719,233.249,-66.123,-177.740,7.734,148.822
C01541=1144.723,233.000,-66.097,-177.744,7.732,148.822
C01542=1144.727,232.752,-66.070,-177.747,7.729,148.822
C01543=1144.732,232.503,-66.044,-177.749,7.726,148.822
C01544=1144.737,232.256,-66.018,-177.752,7.724,148.822
C01545=1144.742,232.007,-65.992,-177.754,7.721,148.822
C01546=1144.746,231.758,-65.965,-177.757,7.718,148.822
C01547=1144.750,231.510,-65.939,-177.760,7.715,148.822
C01548=1144.755,231.260,-65.913,-177.763,7.712,148.823
C01549=1144.759,231.012,-65.887,-177.766,7.709,148.823
C01550=1144.764,230.763,-65.860,-177.769,7.706,148.823
C01551=1144.768,230.515,-65.834,-177.771,7.704,148.823
C01552=1144.772,230.266,-65.808,-177.774,7.701,148.823
C01553=1144.777,230.018,-65.782,-177.777,7.698,148.823
C01554=1144.781,229.770,-65.756,-177.779,7.696,148.823
C01555=1144.786,229.521,-65.730,-177.783,7.693,148.824
C01556=1144.791,229.272,-65.704,-177.785,7.690,148.824
C01557=1144.794,229.023,-65.677,-177.788,7.687,148.824
C01558=1144.799,228.775,-65.651,-177.790,7.685,148.824
C01559=1144.804,228.526,-65.625,-177.793,7.682,148.824
C01560=1144.808,228.278,-65.599,-177.796,7.679,148.824
C01561=1144.812,228.029,-65.573,-177.799,7.676,148.824
C01562=1144.817,227.780,-65.547,-177.802,7.674,148.824
C01563=1144.822,227.531,-65.521,-177.805,7.671,148.825
C01564=1144.826,227.283,-65.495,-177.807,7.669,148.825
C01565=1144.830,227.035,-65.469,-177.810,7.666,148.825
C01566=1144.835,226.786,-65.443,-177.813,7.663,148.825
C01567=1144.839,226.537,-65.418,-177.816,7.660,148.825
C01568=1144.844,226.288,-65.391,-177.819,7.657,148.825
C01569=1144.849,226.040,-65.366,-177.822,7.654,148.825
C01570=1144.853,225.791,-65.340,-177.824,7.652,148.825
C01571=1144.857,225.543,-65.314,-177.827,7.649,148.826
C01572=1144.861,225.294,-65.288,-177.830,7.647,148.826
C01573=1144.866,225.045,-65.262,-177.833,7.644,148.826
C01574=1144.871,224.797,-65.236,-177.835,7.641,148.826
C01575=1144.875,224.548,-65.210,-177.838,7.639,148.826
C01576=1144.879,224.300,-65.185,-177.840,7.636,148.826
C01577=1144.884,224.051,-65.159,-177.844,7.633,148.826
C01578=1144.888,223.803,-65.134,-177.846,7.631,148.827
C01579=1144.892,223.554,-65.108,-177.849,7.628,148.827
C01580=1144.897,223.305,-65.081,-177.851,7.626,148.827
C01581=1144.902,223.057,-65.056,-177.854,7.623,148.827
C01582=1144.906,222.808,-65.030,-177.857,7.620,148.827
C01583=1144.911,222.559,-65.005,-177.860,7.617,148.827
C01584=1144.916,222.311,-64.979,-177.863,7.614,148.827
C01585=1144.920,222.062,-64.953,-177.865,7.612,148.828
C01586=1144.924,221.813,-64.928,-177.869,7.610,148.828
C01587=1144.929,221.565,-64.902,-177.871,7.607,148.828
C01588=1144.933,221.316,-64.877,-177.874,7.604,148.828
C01589=1144.937,221.068,-64.851,-177.876,7.602,148.828
C01590=1144.942,220.819,-64.826,-177.879,7.599,148.828
C01591=1144.947,220.570,-64.800,-177.882,7.596,148.829
C01592=1144.951,220.321,-64.775,-177.885,7.593,148.829
C01593=1144.956,220.073,-64.749,-177.888,7.590,148.829
C01594=1144.960,219.824,-64.724,-177.890,7.588,148.829
C01595=1144.964,219.576,-64.698,-177.894,7.586,148.829
C01596=1144.969,219.327,-64.673,-177.896,7.583,148.829
C01597=1144.973,219.078,-64.647,-177.899,7.580,148.829
C01598=1144.978,218.829,-64.622,-177.901,7.578,148.829
C01599=1144.983,218.581,-64.596,-177.905,7.575,148.830
C01600=1144.987,218.332,-64.570,-177.907,7.572,148.830
C01601=1144.992,218.084,-64.546,-177.910,7.569,148.830
C01602=1144.996,217.835,-64.520,-177.912,7.567,148.830
C01603=1145.000,217.586,-64.494,-177.916,7.565,148.830
C01604=1145.005,217.338,-64.470,-177.918,7.562,148.830
C01605=1145.009,217.089,-64.444,-177.921,7.559,148.831
C01606=1145.014,216.841,-64.419,-177.924,7.557,148.831
C01607=1145.018,216.591,-64.394,-177.927,7.554,148.831
C01608=1145.023,216.342,-64.368,-177.930,7.551,148.831
C01609=1145.027,216.094,-64.343,-177.932,7.548,148.831
C01610=1145.032,215.845,-64.318,-177.935,7.547,148.832
C01611=1145.036,215.597,-64.293,-177.938,7.544,148.832
C01612=1145.040,215.348,-64.268,-177.941,7.541,148.832
C01613=1145.045,215.100,-64.243,-177.944,7.538,148.832
C01614=1145.050,214.851,-64.217,-177.946,7.536,148.832
C01615=1145.055,214.602,-64.192,-177.949,7.533,148.832
C01616=1145.058,214.354,-64.167,-177.952,7.530,148.832
C01617=1145.063,214.105,-64.142,-177.955,7.528,148.833
C01618=1145.068,213.856,-64.117,-177.957,7.526,148.833
C01619=1145.072,213.607,-64.092,-177.960,7.523,148.833
C01620=1145.077,213.359,-64.066,-177.963,7.520,148.833
C01621=1145.081,213.109,-64.042,-177.965,7.518,148.833
C01622=1145.085,212.861,-64.016,-177.968,7.515,148.833
C01623=1145.091,212.613,-63.992,-177.972,7.513,148.834
C01624=1145.095,212.364,-63.966,-177.974,7.510,148.834
C01625=1145.099,212.115,-63.942,-177.977,7.508,148.834
C01626=1145.104,211.866,-63.917,-177.980,7.505,148.834
C01627=1145.109,211.618,-63.892,-177.983,7.502,148.834
C01628=1145.112,211.369,-63.867,-177.985,7.500,148.835
C01629=1145.118,211.120,-63.842,-177.988,7.497,148.835
C01630=1145.122,210.871,-63.817,-177.991,7.494,148.835
C01631=1145.126,210.623,-63.793,-177.993,7.492,148.835
C01632=1145.130,210.374,-63.767,-177.996,7.490,148.835
C01633=1145.135,210.125,-63.742,-177.999,7.487,148.835
C01634=1145.140,209.854,-63.715,-178.002,7.484,148.836
C01635=1145.145,209.584,-63.688,-178.005,7.481,148.836
C01636=1145.150,209.313,-63.661,-178.008,7.478,148.836
C01637=1145.155,209.043,-63.635,-178.011,7.476,148.836
C01638=1145.159,208.794,-63.610,-178.014,7.473,148.836
C01639=1145.164,208.545,-63.585,-178.017,7.471,148.837
C01640=1145.169,208.297,-63.560,-178.020,7.468,148.837
C01641=1145.173,208.048,-63.535,-178.022,7.465,148.837
C01642=1145.178,207.799,-63.511,-178.025,7.464,148.837
C01643=1145.182,207.550,-63.486,-178.028,7.461,148.837
C01644=1145.187,207.302,-63.462,-178.031,7.458,148.838
C01645=1145.192,207.053,-63.437,-178.033,7.456,148.838
C01646=1145.195,206.804,-63.412,-178.036,7.453,148.838
C01647=1145.200,206.556,-63.387,-178.039,7.451,148.838
C01648=1145.205,206.307,-63.363,-178.042,7.449,148.838
C01649=1145.209,206.058,-63.338,-178.044,7.446,148.839
C01650=1145.214,205.809,-63.314,-178.048,7.443,148.839
C01651=1145.219,205.561,-63.290,-178.050,7.441,148.839
C01652=1145.223,205.311,-63.264,-178.053,7.438,148.839
C01653=1145.228,205.063,-63.240,-178.056,7.436,148.839
C01654=1145.233,204.814,-63.216,-178.058,7.433,148.840
C01655=1145.237,204.565,-63.191,-178.061,7.431,148.840
C01656=1145.241,204.317,-63.167,-178.064,7.428,148.840
C01657=1145.246,204.068,-63.143,-178.067,7.426,148.840
C01658=1145.250,203.819,-63.118,-178.070,7.423,148.840
C01659=1145.255,203.570,-63.093,-178.072,7.421,148.841
C01660=1145.259,203.322,-63.069,-178.075,7.419,148.841
C01661=1145.265,203.073,-63.045,-178.078,7.416,148.841
C01662=1145.268,202.824,-63.020,-178.081,7.414,148.841
C01663=1145.273,202.575,-62.996,-178.084,7.411,148.841
C01664=1145.278,202.327,-62.972,-178.086,7.408,148.842
C01665=1145.282,202.077,-62.947,-178.089,7.406,148.842
C01666=1145.286,201.829,-62.923,-178.092,7.404,148.842
C01667=1145.291,201.580,-62.898,-178.095,7.401,148.842
C01668=1145.296,201.332,-62.874,-178.097,7.399,148.842
C01669=1145.300,201.082,-62.850,-178.101,7.396,148.843
C01670=1145.305,200.833,-62.826,-178.103,7.394,148.843
C01671=1145.309,200.585,-62.802,-178.106,7.392,148.843
C01672=1145.314,200.337,-62.778,-178.109,7.389,148.843
C01673=1145.319,200.088,-62.753,-178.111,7.387,148.843
C01674=1145.323,199.839,-62.729,-178.114,7.384,148.844
C01675=1145.327,199.590,-62.705,-178.117,7.382,148.844
C01676=1145.332,199.341,-62.681,-178.120,7.379,148.844
C01677=1145.337,199.093,-62.657,-178.123,7.377,148.844
C01678=1145.341,198.844,-62.632,-178.125,7.375,148.845
C01679=1145.345,198.594,-62.609,-178.128,7.372,148.845
C01680=1145.350,198.346,-62.584,-178.131,7.369,148.845
C01681=1145.355,198.097,-62.560,-178.134,7.367,148.845
C01682=1145.359,197.848,-62.537,-178.137,7.365,148.846
C01683=1145.364,197.600,-62.513,-178.139,7.363,148.846
C01684=1145.368,197.350,-62.487,-178.142,7.360,148.846
C01685=1145.373,197.101,-62.464,-178.145,7.358,148.846
C01686=1145.377,196.853,-62.440,-178.147,7.355,148.846
C01687=1145.382,196.605,-62.416,-178.151,7.352,148.847
C01688=1145.387,196.356,-62.393,-178.153,7.350,148.847
C01689=1145.392,196.107,-62.368,-178.156,7.348,148.847
C01690=1145.396,195.858,-62.344,-178.158,7.346,148.847
C01691=1145.400,195.609,-62.320,-178.162,7.343,148.848
C01692=1145.405,195.360,-62.296,-178.165,7.340,148.848
C01693=1145.409,195.111,-62.273,-178.167,7.339,148.848
C01694=1145.414,194.863,-62.249,-178.170,7.336,148.848
C01695=1145.419,194.614,-62.225,-178.173,7.334,148.849
C01696=1145.424,194.365,-62.201,-178.176,7.331,148.849
C01697=1145.428,194.116,-62.177,-178.178,7.329,148.849
C01698=1145.433,193.868,-62.153,-178.181,7.326,148.849
C01699=1145.437,193.619,-62.130,-178.184,7.324,148.849
C01700=1145.442,193.370,-62.106,-178.187,7.322,148.850
C01701=1145.446,193.121,-62.082,-178.190,7.319,148.850
C01702=1145.450,192.872,-62.058,-178.192,7.317,148.850
C01703=1145.455,192.623,-62.035,-178.195,7.314,148.850
C01704=1145.460,192.374,-62.011,-178.198,7.312,148.851
C01705=1145.464,192.126,-61.987,-178.201,7.310,148.851
C01706=1145.469,191.877,-61.964,-178.203,7.308,148.851
C01707=1145.473,191.628,-61.940,-178.206,7.305,148.851
C01708=1145.478,191.379,-61.916,-178.210,7.303,148.852
C01709=1145.482,191.130,-61.893,-178.212,7.301,148.852
C01710=1145.487,190.882,-61.869,-178.215,7.298,148.852
C01711=1145.492,190.633,-61.846,-178.217,7.296,148.852
C01712=1145.496,190.384,-61.822,-178.221,7.293,148.853
C01713=1145.501,190.135,-61.798,-178.223,7.291,148.853
C01714=1145.505,189.886,-61.775,-178.226,7.289,148.853
C01715=1145.510,189.637,-61.751,-178.228,7.287,148.853
C01716=1145.515,189.388,-61.728,-178.232,7.284,148.854
C01717=1145.519,189.140,-61.704,-178.234,7.282,148.854
C01718=1145.524,188.891,-61.681,-178.237,7.279,148.854
C01719=1145.529,188.642,-61.657,-178.240,7.278,148.854
C01720=1145.533,188.393,-61.634,-178.243,7.275,148.855
C01721=1145.538,188.144,-61.610,-178.245,7.273,148.855
C01722=1145.542,187.895,-61.586,-178.248,7.270,148.855
C01723=1145.547,187.646,-61.563,-178.251,7.268,148.855
C01724=1145.552,187.397,-61.540,-178.254,7.265,148.855
C01725=1145.556,187.148,-61.516,-178.257,7.263,148.856
C01726=1145.562,186.900,-61.493,-178.259,7.261,148.856
C01727=1145.566,186.651,-61.471,-178.262,7.258,148.856
C01728=1145.570,186.403,-61.447,-178.265,7.257,148.857
C01729=1145.575,186.154,-61.423,-178.268,7.254,148.857
C01730=1145.580,185.905,-61.400,-178.271,7.252,148.857
C01731=1145.584,185.655,-61.377,-178.273,7.249,148.857
C01732=1145.589,185.406,-61.353,-178.276,7.247,148.858
C01733=1145.593,185.158,-61.330,-178.279,7.245,148.858
C01734=1145.598,184.909,-61.307,-178.282,7.243,148.858
C01735=1145.602,184.660,-61.284,-178.285,7.240,148.858
C01736=1145.607,184.411,-61.260,-178.287,7.238,148.859
C01737=1145.612,184.162,-61.237,-178.290,7.235,148.859
C01738=1145.616,183.892,-61.213,-178.293,7.234,148.859
C01739=1145.621,183.623,-61.187,-178.296,7.231,148.859
C01740=1145.627,183.353,-61.162,-178.299,7.228,148.860
C01741=1145.632,183.083,-61.137,-178.302,7.226,148.860
C01742=1145.636,182.835,-61.114,-178.305,7.224,148.860
C01743=1145.641,182.586,-61.091,-178.308,7.221,148.861
C01744=1145.645,182.337,-61.067,-178.311,7.219,148.861
C01745=1145.650,182.089,-61.045,-178.313,7.216,148.861
C01746=1145.655,181.840,-61.021,-178.316,7.215,148.861
C01747=1145.660,181.590,-60.999,-178.319,7.213,148.862
C01748=1145.663,181.341,-60.976,-178.322,7.210,148.862
C01749=1145.668,181.092,-60.953,-178.324,7.208,148.862
C01750=1145.673,180.843,-60.929,-178.327,7.205,148.862
C01751=1145.677,180.595,-60.907,-178.330,7.204,148.863
C01752=1145.682,180.346,-60.884,-178.333,7.201,148.863
C01753=1145.687,180.096,-60.861,-178.335,7.199,148.863
C01754=1145.691,179.848,-60.838,-178.339,7.197,148.864
C01755=1145.696,179.599,-60.815,-178.341,7.195,148.864
C01756=1145.701,179.350,-60.792,-178.344,7.192,148.864
C01757=1145.705,179.102,-60.769,-178.347,7.190,148.864
C01758=1145.710,178.852,-60.746,-178.349,7.188,148.865
C01759=1145.714,178.603,-60.724,-178.352,7.186,148.865
C01760=1145.719,178.355,-60.701,-178.355,7.184,148.865
C01761=1145.724,178.105,-60.678,-178.358,7.181,148.865
C01762=1145.728,177.857,-60.655,-178.360,7.179,148.866
C01763=1145.733,177.608,-60.632,-178.364,7.177,148.866
C01764=1145.738,177.359,-60.610,-178.366,7.175,148.866
C01765=1145.743,177.110,-60.587,-178.369,7.172,148.867
C01766=1145.747,176.861,-60.564,-178.372,7.170,148.867
C01767=1145.752,176.612,-60.541,-178.374,7.168,148.867
C01768=1145.756,176.364,-60.519,-178.377,7.166,148.867
C01769=1145.761,176.114,-60.496,-178.380,7.164,148.868
C01770=1145.765,175.865,-60.474,-178.383,7.161,148.868
C01771=1145.770,175.616,-60.450,-178.386,7.159,148.868
C01772=1145.775,175.367,-60.429,-178.389,7.157,148.869
C01773=1145.779,175.118,-60.405,-178.391,7.155,148.869
C01774=1145.784,174.869,-60.383,-178.394,7.153,148.869
C01775=1145.789,174.621,-60.360,-178.397,7.150,148.870
C01776=1145.793,174.372,-60.337,-178.399,7.148,148.870
C01777=1145.798,174.122,-60.315,-178.403,7.146,148.870
C01778=1145.802,173.874,-60.292,-178.405,7.144,148.870
C01779=1145.807,173.625,-60.270,-178.408,7.142,148.871
C01780=1145.812,173.375,-60.248,-178.411,7.139,148.871
C01781=1145.816,173.127,-60.225,-178.414,7.138,148.871
C01782=1145.821,172.878,-60.203,-178.417,7.135,148.872
C01783=1145.825,172.629,-60.180,-178.419,7.133,148.872
C01784=1145.831,172.380,-60.158,-178.422,7.131,148.872
C01785=1145.835,172.131,-60.135,-178.425,7.129,148.872
C01786=1145.839,171.882,-60.113,-178.427,7.127,148.873
C01787=1145.845,171.633,-60.091,-178.431,7.124,148.873
C01788=1145.849,171.384,-60.068,-178.433,7.122,148.873
C01789=1145.854,171.135,-60.045,-178.436,7.121,148.874
C01790=1145.858,170.887,-60.023,-178.439,7.118,148.874
C01791=1145.863,170.637,-60.001,-178.442,7.116,148.874
C01792=1145.868,170.388,-59.978,-178.445,7.113,148.875
C01793=1145.872,170.140,-59.956,-178.447,7.111,148.875
C01794=1145.877,169.891,-59.934,-178.450,7.110,148.875
C01795=1145.881,169.642,-59.912,-178.453,7.107,148.875
C01796=1145.887,169.393,-59.890,-178.456,7.105,148.876
C01797=1145.891,169.144,-59.867,-178.458,7.103,148.876
C01798=1145.895,168.895,-59.845,-178.461,7.101,148.876
C01799=1145.901,168.646,-59.823,-178.464,7.099,148.877
C01800=1145.905,168.396,-59.800,-178.467,7.096,148.877
C01801=1145.909,168.148,-59.778,-178.469,7.094,148.877
C01802=1145.914,167.899,-59.756,-178.472,7.093,148.878
C01803=1145.919,167.650,-59.734,-178.475,7.090,148.878
C01804=1145.924,167.401,-59.712,-178.478,7.088,148.878
C01805=1145.928,167.152,-59.690,-178.480,7.086,148.878
C01806=1145.932,166.903,-59.667,-178.484,7.084,148.879
